C07133=1014.143,341.279,-151.610,170.583,52.042,160.243
C07134=1014.136,341.031,-151.575,170.576,52.047,160.243
C07135=1014.129,340.783,-151.540,170.568,52.051,160.243
C07136=1014.122,340.536,-151.504,170.561,52.056,160.242
C07137=1014.116,340.289,-151.469,170.554,52.060,160.242
C07138=1014.109,340.041,-151.433,170.546,52.065,160.241
C07139=1014.103,339.794,-151.398,170.539,52.069,160.241
C07140=1014.095,339.546,-151.362,170.530,52.073,160.240
C07141=1014.088,339.299,-151.326,170.523,52.077,160.240
C07142=1014.081,339.052,-151.291,170.515,52.082,160.240
C07143=1014.075,338.805,-151.256,170.508,52.086,160.239
C07144=1014.067,338.513,-151.215,170.499,52.092,160.239
C07145=1014.059,338.221,-151.173,170.490,52.097,160.239
C07146=1014.052,337.930,-151.132,170.481,52.103,160.238
C07147=1014.044,337.638,-151.090,170.472,52.108,160.238
C07148=1014.036,337.391,-151.056,170.465,52.112,160.237
C07149=1014.029,337.143,-151.021,170.457,52.117,160.237
C07150=1014.022,336.896,-150.986,170.450,52.122,160.237
C07151=1014.016,336.648,-150.951,170.442,52.127,160.236
C07152=1014.009,336.401,-150.916,170.435,52.131,160.236
C07153=1014.002,336.153,-150.881,170.426,52.136,160.236
C07154=1013.996,335.906,-150.846,170.420,52.141,160.236
C07155=1013.989,335.658,-150.811,170.412,52.146,160.235
C07156=1013.983,335.410,-150.776,170.405,52.150,160.235
C07157=1013.976,335.163,-150.741,170.397,52.154,160.234
C07158=1013.969,334.915,-150.707,170.390,52.160,160.234
C07159=1013.963,334.668,-150.672,170.383,52.164,160.234
C07160=1013.956,334.421,-150.637,170.374,52.169,160.233
C07161=1013.949,334.173,-150.603,170.368,52.174,160.233
C07162=1013.942,333.926,-150.568,170.361,52.178,160.233
C07163=1013.936,333.678,-150.533,170.353,52.183,160.233
C07164=1013.929,333.431,-150.498,170.346,52.188,160.232
C07165=1013.923,333.183,-150.464,170.338,52.192,160.232
C07166=1013.917,332.936,-150.429,170.331,52.197,160.232
C07167=1013.910,332.688,-150.395,170.324,52.202,160.232
C07168=1013.903,332.441,-150.359,170.316,52.207,160.231
C07169=1013.897,332.193,-150.325,170.309,52.211,160.231
C07170=1013.891,331.945,-150.291,170.301,52.217,160.231
C07171=1013.883,331.698,-150.256,170.294,52.221,160.230
C07172=1013.877,331.450,-150.222,170.287,52.226,160.230
C07173=1013.871,331.203,-150.188,170.280,52.231,160.230
C07174=1013.864,330.955,-150.154,170.272,52.236,160.230
C07175=1013.857,330.707,-150.120,170.265,52.241,160.230
C07176=1013.851,330.460,-150.085,170.258,52.246,160.229
C07177=1013.844,330.213,-150.051,170.251,52.251,160.229
C07178=1013.838,329.965,-150.017,170.243,52.256,160.229
C07179=1013.831,329.717,-149.982,170.236,52.261,160.229
C07180=1013.825,329.470,-149.949,170.229,52.266,160.229
C07181=1013.818,329.222,-149.914,170.222,52.271,160.228
C07182=1013.812,328.975,-149.881,170.215,52.276,160.228
C07183=1013.805,328.727,-149.847,170.207,52.281,160.228
C07184=1013.799,328.479,-149.812,170.201,52.286,160.228
C07185=1013.792,328.232,-149.779,170.194,52.291,160.228
C07186=1013.786,327.984,-149.744,170.186,52.296,160.227
C07187=1013.780,327.737,-149.710,170.179,52.301,160.227
C07188=1013.772,327.489,-149.676,170.171,52.306,160.227
C07189=1013.767,327.242,-149.642,170.165,52.311,160.227
C07190=1013.760,326.994,-149.608,170.158,52.316,160.227
C07191=1013.754,326.746,-149.575,170.150,52.322,160.226
C07192=1013.747,326.498,-149.541,170.143,52.327,160.226
C07193=1013.742,326.251,-149.507,170.137,52.332,160.226
C07194=1013.734,326.003,-149.473,170.129,52.337,160.226
C07195=1013.728,325.756,-149.439,170.122,52.342,160.226
C07196=1013.722,325.508,-149.406,170.116,52.347,160.226
C07197=1013.715,325.261,-149.372,170.108,52.352,160.225
C07198=1013.709,325.013,-149.339,170.101,52.357,160.225
C07199=1013.702,324.765,-149.305,170.093,52.363,160.225
C07200=1013.696,324.518,-149.272,170.087,52.368,160.225
C07201=1013.689,324.270,-149.239,170.080,52.374,160.225
C07202=1013.682,324.022,-149.206,170.073,52.379,160.225
C07203=1013.676,323.775,-149.171,170.066,52.384,160.225
C07204=1013.669,323.479,-149.132,170.058,52.390,160.224
C07205=1013.660,323.183,-149.093,170.050,52.397,160.224
C07206=1013.653,322.887,-149.053,170.040,52.404,160.224
C07207=1013.645,322.591,-149.013,170.032,52.410,160.224
C07208=1013.638,322.344,-148.980,170.025,52.415,160.224
C07209=1013.632,322.096,-148.947,170.019,52.421,160.224
C07210=1013.626,321.848,-148.913,170.011,52.426,160.224
C07211=1013.620,321.600,-148.880,170.005,52.431,160.224
C07212=1013.613,321.353,-148.847,169.998,52.437,160.224
C07213=1013.606,321.105,-148.814,169.991,52.442,160.224
C07214=1013.600,320.857,-148.781,169.984,52.448,160.224
C07215=1013.594,320.609,-148.748,169.977,52.453,160.223
C07216=1013.588,320.362,-148.715,169.970,52.458,160.223
C07217=1013.581,320.113,-148.682,169.964,52.464,160.223
C07218=1013.575,319.866,-148.649,169.956,52.469,160.223
C07219=1013.568,319.619,-148.616,169.950,52.475,160.223
C07220=1013.563,319.371,-148.582,169.943,52.480,160.223
C07221=1013.556,319.123,-148.550,169.936,52.486,160.223
C07222=1013.550,318.876,-148.517,169.929,52.491,160.223
C07223=1013.544,318.628,-148.484,169.922,52.497,160.223
C07224=1013.537,318.380,-148.451,169.916,52.503,160.223
C07225=1013.531,318.132,-148.418,169.909,52.508,160.223
C07226=1013.525,317.884,-148.385,169.902,52.514,160.223
C07227=1013.519,317.637,-148.352,169.895,52.519,160.223
C07228=1013.513,317.389,-148.320,169.889,52.525,160.223
C07229=1013.506,317.142,-148.287,169.881,52.531,160.223
C07230=1013.500,316.894,-148.254,169.875,52.536,160.223
C07231=1013.494,316.646,-148.221,169.869,52.542,160.223
C07232=1013.488,316.398,-148.189,169.861,52.548,160.223
C07233=1013.482,316.150,-148.156,169.855,52.553,160.223
C07234=1013.476,315.903,-148.123,169.848,52.558,160.223
C07235=1013.470,315.655,-148.090,169.841,52.564,160.223
C07236=1013.464,315.407,-148.057,169.835,52.570,160.223
C07237=1013.458,315.159,-148.025,169.829,52.576,160.223
C07238=1013.452,314.911,-147.992,169.821,52.581,160.223
C07239=1013.445,314.664,-147.960,169.815,52.587,160.223
C07240=1013.439,314.416,-147.927,169.808,52.593,160.223
C07241=1013.433,314.168,-147.895,169.801,52.599,160.223
C07242=1013.428,313.920,-147.861,169.795,52.605,160.223
C07243=1013.422,313.673,-147.829,169.788,52.610,160.223
C07244=1013.416,313.425,-147.797,169.781,52.616,160.223
C07245=1013.410,313.177,-147.764,169.775,52.621,160.223
C07246=1013.403,312.930,-147.732,169.768,52.627,160.223
C07247=1013.397,312.682,-147.700,169.761,52.633,160.223
C07248=1013.392,312.434,-147.666,169.755,52.639,160.223
C07249=1013.386,312.186,-147.635,169.749,52.645,160.223
C07250=1013.380,311.939,-147.602,169.741,52.651,160.223
C07251=1013.374,311.691,-147.569,169.735,52.656,160.223
C07252=1013.368,311.443,-147.537,169.729,52.662,160.223
C07253=1013.363,311.196,-147.504,169.723,52.668,160.223
C07254=1013.357,310.947,-147.472,169.715,52.674,160.223
C07255=1013.351,310.700,-147.439,169.709,52.680,160.223
C07256=1013.345,310.452,-147.407,169.703,52.685,160.223
C07257=1013.339,310.204,-147.376,169.696,52.691,160.223
C07258=1013.333,309.956,-147.343,169.689,52.697,160.223
C07259=1013.328,309.708,-147.310,169.683,52.703,160.223
C07260=1013.322,309.461,-147.278,169.676,52.709,160.223
C07261=1013.316,309.213,-147.246,169.670,52.715,160.224
C07262=1013.310,308.965,-147.214,169.664,52.721,160.224
C07263=1013.304,308.717,-147.183,169.657,52.727,160.224
C07264=1013.297,308.427,-147.145,169.650,52.734,160.224
C07265=1013.290,308.137,-147.109,169.642,52.741,160.224
C07266=1013.283,307.846,-147.071,169.634,52.748,160.224
C07267=1013.275,307.555,-147.034,169.627,52.756,160.225
C07268=1013.269,307.308,-147.003,169.621,52.762,160.225
C07269=1013.263,307.060,-146.971,169.613,52.768,160.225
C07270=1013.257,306.812,-146.939,169.607,52.774,160.225
C07271=1013.251,306.564,-146.908,169.600,52.781,160.225
C07272=1013.245,306.316,-146.876,169.594,52.787,160.225
C07273=1013.239,306.069,-146.845,169.588,52.793,160.225
C07274=1013.233,305.820,-146.814,169.581,52.799,160.225
C07275=1013.227,305.573,-146.782,169.575,52.805,160.225
C07276=1013.221,305.325,-146.750,169.568,52.812,160.226
C07277=1013.214,305.077,-146.719,169.562,52.818,160.226
C07278=1013.209,304.829,-146.688,169.556,52.824,160.226
C07279=1013.202,304.581,-146.657,169.549,52.830,160.226
C07280=1013.197,304.333,-146.625,169.543,52.837,160.226
C07281=1013.190,304.085,-146.594,169.536,52.843,160.226
C07282=1013.185,303.837,-146.563,169.530,52.849,160.227
C07283=1013.178,303.589,-146.531,169.524,52.856,160.227
C07284=1013.173,303.342,-146.499,169.517,52.862,160.227
C07285=1013.167,303.093,-146.469,169.511,52.868,160.227
C07286=1013.161,302.846,-146.437,169.505,52.875,160.227
C07287=1013.155,302.597,-146.406,169.498,52.881,160.227
C07288=1013.149,302.350,-146.375,169.493,52.887,160.228
C07289=1013.144,302.102,-146.344,169.486,52.894,160.228
C07290=1013.138,301.854,-146.312,169.480,52.900,160.228
C07291=1013.131,301.607,-146.281,169.474,52.906,160.228
C07292=1013.126,301.358,-146.250,169.467,52.913,160.228
C07293=1013.120,301.110,-146.218,169.461,52.919,160.229
C07294=1013.115,300.862,-146.188,169.454,52.926,160.229
C07295=1013.109,300.614,-146.157,169.448,52.932,160.229
C07296=1013.103,300.366,-146.126,169.442,52.938,160.229
C07297=1013.098,300.118,-146.095,169.436,52.945,160.230
C07298=1013.091,299.870,-146.063,169.430,52.952,160.230
C07299=1013.086,299.622,-146.032,169.423,52.958,160.230
C07300=1013.080,299.374,-146.002,169.417,52.964,160.230
C07301=1013.074,299.126,-145.970,169.411,52.971,160.230
C07302=1013.068,298.878,-145.940,169.404,52.977,160.231
C07303=1013.063,298.631,-145.908,169.398,52.984,160.231
C07304=1013.057,298.383,-145.878,169.393,52.990,160.231
C07305=1013.051,298.134,-145.846,169.386,52.997,160.231
C07306=1013.046,297.886,-145.816,169.380,53.004,160.232
C07307=1013.040,297.639,-145.784,169.373,53.010,160.232
C07308=1013.034,297.391,-145.754,169.368,53.017,160.232
C07309=1013.029,297.142,-145.723,169.362,53.023,160.232
C07310=1013.023,296.894,-145.692,169.355,53.030,160.233
C07311=1013.017,296.647,-145.661,169.349,53.037,160.233
C07312=1013.012,296.399,-145.630,169.344,53.043,160.233
C07313=1013.007,296.151,-145.599,169.337,53.050,160.233
C07314=1013.000,295.902,-145.569,169.331,53.056,160.234
C07315=1012.995,295.654,-145.538,169.325,53.063,160.234
C07316=1012.989,295.406,-145.507,169.318,53.070,160.234
C07317=1012.984,295.158,-145.476,169.313,53.076,160.234
C07318=1012.978,294.911,-145.446,169.306,53.083,160.235
C07319=1012.973,294.663,-145.414,169.300,53.089,160.235
C07320=1012.967,294.415,-145.384,169.294,53.096,160.235
C07321=1012.962,294.167,-145.353,169.288,53.103,160.235
C07322=1012.956,293.919,-145.323,169.282,53.109,160.236
C07323=1012.951,293.671,-145.292,169.276,53.116,160.236
C07324=1012.945,293.398,-145.258,169.269,53.123,160.236
C07325=1012.939,293.126,-145.224,169.262,53.131,160.237
C07326=1012.933,292.853,-145.190,169.256,53.138,160.237
C07327=1012.927,292.582,-145.157,169.249,53.145,160.237
C07328=1012.922,292.334,-145.126,169.243,53.153,160.238
C07329=1012.916,292.085,-145.097,169.237,53.159,160.238
C07330=1012.911,291.837,-145.066,169.231,53.166,160.238
C07331=1012.905,291.590,-145.036,169.225,53.173,160.239
C07332=1012.899,291.342,-145.006,169.219,53.180,160.239
C07333=1012.894,291.093,-144.976,169.213,53.187,160.239
C07334=1012.888,290.845,-144.945,169.207,53.194,160.240
C07335=1012.883,290.597,-144.915,169.200,53.201,160.240
C07336=1012.877,290.349,-144.885,169.195,53.208,160.240
C07337=1012.871,290.101,-144.855,169.189,53.214,160.241
C07338=1012.866,289.853,-144.825,169.183,53.222,160.241
C07339=1012.860,289.605,-144.795,169.177,53.228,160.241
C07340=1012.854,289.356,-144.765,169.171,53.236,160.242
C07341=1012.849,289.109,-144.735,169.165,53.242,160.242
C07342=1012.843,288.860,-144.705,169.159,53.250,160.242
C07343=1012.837,288.612,-144.675,169.153,53.256,160.243
C07344=1012.832,288.364,-144.645,169.147,53.264,160.243
C07345=1012.826,288.115,-144.616,169.141,53.270,160.243
C07346=1012.821,287.868,-144.586,169.135,53.278,160.244
C07347=1012.816,287.620,-144.556,169.130,53.285,160.244
C07348=1012.810,287.372,-144.526,169.124,53.292,160.245
C07349=1012.804,287.124,-144.496,169.118,53.299,160.245
C07350=1012.799,286.875,-144.466,169.112,53.306,160.245
C07351=1012.793,286.627,-144.436,169.105,53.313,160.246
C07352=1012.787,286.379,-144.406,169.100,53.320,160.246
C07353=1012.782,286.131,-144.377,169.094,53.328,160.247
C07354=1012.777,285.883,-144.347,169.088,53.334,160.247
C07355=1012.771,285.635,-144.317,169.082,53.342,160.247
C07356=1012.766,285.386,-144.287,169.077,53.349,160.248
C07357=1012.760,285.138,-144.258,169.070,53.356,160.248
C07358=1012.755,284.890,-144.229,169.065,53.363,160.248
C07359=1012.750,284.642,-144.199,169.058,53.371,160.249
C07360=1012.744,284.393,-144.169,169.053,53.378,160.249
C07361=1012.738,284.146,-144.139,169.047,53.385,160.250
C07362=1012.733,283.898,-144.110,169.041,53.392,160.250
C07363=1012.727,283.650,-144.081,169.035,53.400,160.250
C07364=1012.722,283.401,-144.051,169.029,53.407,160.251
C07365=1012.717,283.154,-144.022,169.023,53.414,160.251
C07366=1012.711,282.905,-143.993,169.018,53.421,160.252
C07367=1012.705,282.657,-143.963,169.012,53.429,160.252
C07368=1012.700,282.408,-143.934,169.006,53.436,160.253
C07369=1012.694,282.160,-143.905,169.000,53.444,160.253
C07370=1012.689,281.912,-143.876,168.995,53.451,160.254
C07371=1012.683,281.664,-143.846,168.988,53.459,160.254
C07372=1012.678,281.416,-143.817,168.983,53.466,160.255
C07373=1012.672,281.168,-143.788,168.977,53.473,160.255
C07374=1012.666,280.919,-143.758,168.972,53.481,160.255
C07375=1012.662,280.671,-143.730,168.965,53.488,160.256
C07376=1012.656,280.423,-143.701,168.960,53.495,160.256
C07377=1012.651,280.175,-143.671,168.954,53.503,160.257
C07378=1012.645,279.927,-143.642,168.948,53.510,160.257
C07379=1012.640,279.678,-143.613,168.942,53.518,160.258
C07380=1012.634,279.430,-143.584,168.936,53.525,160.258
C07381=1012.629,279.182,-143.555,168.931,53.533,160.259
C07382=1012.624,278.934,-143.525,168.924,53.540,160.259
C07383=1012.618,278.685,-143.497,168.920,53.548,160.260
C07384=1012.612,278.425,-143.466,168.913,53.556,160.260
C07385=1012.607,278.165,-143.435,168.907,53.563,160.260
C07386=1012.602,277.905,-143.405,168.901,53.572,160.261
C07387=1012.596,277.645,-143.374,168.895,53.579,160.261
C07388=1012.587,277.237,-143.328,168.886,53.592,160.262
C07389=1012.579,276.829,-143.280,168.877,53.604,160.263
C07390=1012.570,276.422,-143.232,168.867,53.617,160.264
C07391=1012.561,276.014,-143.184,168.858,53.629,160.265
C07392=1012.347,278.241,-143.809,168.878,53.661,160.276
C07393=1012.354,278.605,-143.851,168.887,53.650,160.276
C07394=1012.362,278.970,-143.893,168.895,53.639,160.275
C07395=1012.370,279.335,-143.936,168.904,53.628,160.274
C07396=1012.379,279.699,-143.979,168.912,53.617,160.274
C07397=1012.383,279.947,-144.008,168.918,53.609,160.273
C07398=1012.389,280.196,-144.037,168.923,53.602,160.273
C07399=1012.394,280.443,-144.066,168.929,53.594,160.272
C07400=1012.400,280.692,-144.096,168.936,53.587,160.272
C07401=1012.404,280.940,-144.124,168.941,53.580,160.271
C07402=1012.410,281.189,-144.154,168.947,53.572,160.271
C07403=1012.416,281.437,-144.183,168.952,53.565,160.270
C07404=1012.421,281.684,-144.212,168.959,53.557,160.270
C07405=1012.426,281.934,-144.241,168.964,53.550,160.270
C07406=1012.433,282.182,-144.270,168.970,53.542,160.269
C07407=1012.437,282.429,-144.299,168.977,53.535,160.269
C07408=1012.443,282.678,-144.329,168.982,53.528,160.268
C07409=1012.448,282.926,-144.359,168.988,53.520,160.268
C07410=1012.454,283.174,-144.387,168.993,53.513,160.267
C07411=1012.460,283.422,-144.417,169.000,53.505,160.267
C07412=1012.465,283.671,-144.447,169.005,53.498,160.266
C07413=1012.471,283.918,-144.475,169.011,53.490,160.266
C07414=1012.476,284.166,-144.505,169.016,53.483,160.266
C07415=1012.482,284.415,-144.534,169.023,53.476,160.265
C07416=1012.487,284.663,-144.564,169.028,53.469,160.265
C07417=1012.492,284.911,-144.593,169.035,53.462,160.264
C07418=1012.498,285.160,-144.623,169.040,53.454,160.264
C07419=1012.503,285.408,-144.653,169.047,53.447,160.264
C07420=1012.508,285.656,-144.682,169.052,53.440,160.263
C07421=1012.514,285.904,-144.712,169.058,53.433,160.263
C07422=1012.519,286.152,-144.742,169.065,53.425,160.263
C07423=1012.525,286.400,-144.772,169.070,53.419,160.262
C07424=1012.530,286.648,-144.801,169.077,53.411,160.262
C07425=1012.535,286.897,-144.830,169.082,53.404,160.261
C07426=1012.541,287.144,-144.861,169.089,53.397,160.261
C07427=1012.547,287.393,-144.890,169.094,53.390,160.261
C07428=1012.552,287.641,-144.920,169.100,53.382,160.260
C07429=1012.558,287.889,-144.950,169.106,53.376,160.260
C07430=1012.563,288.137,-144.980,169.112,53.368,160.260
C07431=1012.568,288.385,-145.009,169.118,53.362,160.259
C07432=1012.574,288.633,-145.040,169.124,53.354,160.259
C07433=1012.580,288.882,-145.069,169.129,53.347,160.258
C07434=1012.585,289.130,-145.099,169.136,53.340,160.258
C07435=1012.591,289.378,-145.129,169.141,53.333,160.258
C07436=1012.597,289.626,-145.159,169.148,53.326,160.258
C07437=1012.602,289.874,-145.189,169.154,53.319,160.257
C07438=1012.607,290.122,-145.219,169.160,53.312,160.257
C07439=1012.613,290.370,-145.249,169.166,53.305,160.256
C07440=1012.619,290.618,-145.279,169.172,53.298,160.256
C07441=1012.625,290.866,-145.309,169.178,53.291,160.256
C07442=1012.630,291.114,-145.339,169.183,53.284,160.255
C07443=1012.635,291.362,-145.369,169.190,53.277,160.255
C07444=1012.641,291.610,-145.400,169.195,53.270,160.255
C07445=1012.646,291.859,-145.429,169.202,53.263,160.254
C07446=1012.652,292.107,-145.460,169.207,53.256,160.254
C07447=1012.658,292.354,-145.490,169.214,53.249,160.254
C07448=1012.663,292.603,-145.521,169.220,53.243,160.253
C07449=1012.669,292.877,-145.555,169.227,53.235,160.253
C07450=1012.676,293.152,-145.588,169.234,53.227,160.253
C07451=1012.681,293.426,-145.622,169.240,53.220,160.253
C07452=1012.688,293.701,-145.656,169.248,53.213,160.252
C07453=1012.693,293.949,-145.687,169.253,53.206,160.252
C07454=1012.699,294.197,-145.717,169.259,53.199,160.251
C07455=1012.704,294.445,-145.748,169.265,53.192,160.251
C07456=1012.710,294.693,-145.779,169.271,53.186,160.251
C07457=1012.715,294.941,-145.810,169.278,53.179,160.251
C07458=1012.720,295.189,-145.840,169.284,53.172,160.251
C07459=1012.726,295.437,-145.871,169.290,53.166,160.250
C07460=1012.731,295.685,-145.901,169.296,53.159,160.250
C07461=1012.736,295.933,-145.932,169.302,53.153,160.250
C07462=1012.742,296.181,-145.963,169.309,53.146,160.250
C07463=1012.747,296.429,-145.994,169.314,53.139,160.249
C07464=1012.754,296.677,-146.024,169.321,53.132,160.249
C07465=1012.759,296.925,-146.056,169.327,53.125,160.249
C07466=1012.765,297.173,-146.086,169.332,53.119,160.248
C07467=1012.770,297.421,-146.117,169.339,53.112,160.248
C07468=1012.775,297.669,-146.148,169.345,53.105,160.248
C07469=1012.781,297.917,-146.179,169.352,53.099,160.248
C07470=1012.787,298.165,-146.211,169.357,53.092,160.247
C07471=1012.793,298.413,-146.241,169.364,53.086,160.247
C07472=1012.798,298.661,-146.272,169.370,53.080,160.247
C07473=1012.804,298.909,-146.302,169.376,53.073,160.247
C07474=1012.810,299.157,-146.334,169.383,53.066,160.247
C07475=1012.815,299.405,-146.365,169.389,53.060,160.246
C07476=1012.820,299.653,-146.396,169.396,53.053,160.246
C07477=1012.827,299.900,-146.427,169.401,53.047,160.246
C07478=1012.832,300.149,-146.458,169.407,53.040,160.246
C07479=1012.838,300.397,-146.488,169.414,53.033,160.245
C07480=1012.843,300.644,-146.520,169.420,53.027,160.245
C07481=1012.850,300.893,-146.551,169.427,53.021,160.245
C07482=1012.855,301.140,-146.582,169.433,53.014,160.245
C07483=1012.861,301.388,-146.613,169.439,53.007,160.245
C07484=1012.867,301.637,-146.644,169.445,53.001,160.244
C07485=1012.873,301.884,-146.675,169.451,52.995,160.244
C07486=1012.878,302.132,-146.706,169.458,52.988,160.244
C07487=1012.885,302.380,-146.737,169.464,52.982,160.244
C07488=1012.890,302.628,-146.768,169.471,52.976,160.244
C07489=1012.897,302.876,-146.800,169.477,52.969,160.244
C07490=1012.902,303.124,-146.831,169.484,52.962,160.243
C07491=1012.908,303.372,-146.862,169.490,52.956,160.243
C07492=1012.914,303.620,-146.894,169.497,52.950,160.243
C07493=1012.920,303.868,-146.924,169.503,52.943,160.243
C07494=1012.926,304.116,-146.956,169.509,52.938,160.243
C07495=1012.932,304.363,-146.987,169.516,52.931,160.243
C07496=1012.937,304.612,-147.019,169.521,52.924,160.242
C07497=1012.943,304.859,-147.050,169.529,52.918,160.242
C07498=1012.949,305.107,-147.082,169.534,52.912,160.242
C07499=1012.955,305.355,-147.113,169.542,52.906,160.242
C07500=1012.961,305.603,-147.144,169.547,52.899,160.242
C07501=1012.967,305.851,-147.176,169.554,52.893,160.242
C07502=1012.973,306.099,-147.207,169.560,52.887,160.242
C07503=1012.979,306.348,-147.238,169.566,52.880,160.241
C07504=1012.985,306.595,-147.270,169.573,52.874,160.241
C07505=1012.991,306.843,-147.302,169.579,52.868,160.241
C07506=1012.997,307.090,-147.333,169.586,52.862,160.241
C07507=1013.003,307.338,-147.365,169.593,52.856,160.241
C07508=1013.010,307.587,-147.395,169.599,52.849,160.241
C07509=1013.016,307.879,-147.434,169.607,52.842,160.241
C07510=1013.024,308.172,-147.470,169.615,52.835,160.241
C07511=1013.031,308.464,-147.507,169.623,52.828,160.240
C07512=1013.038,308.757,-147.544,169.630,52.820,160.240
C07513=1013.044,309.004,-147.577,169.636,52.814,160.240
C07514=1013.050,309.252,-147.609,169.643,52.808,160.240
C07515=1013.056,309.501,-147.641,169.650,52.802,160.240
C07516=1013.061,309.748,-147.673,169.656,52.796,160.240
C07517=1013.068,309.996,-147.705,169.663,52.790,160.240
C07518=1013.072,310.244,-147.738,169.669,52.784,160.240
C07519=1013.079,310.491,-147.770,169.675,52.778,160.240
C07520=1013.085,310.739,-147.802,169.683,52.772,160.240
C07521=1013.090,310.987,-147.834,169.689,52.766,160.240
C07522=1013.096,311.235,-147.867,169.695,52.761,160.239
C07523=1013.102,311.483,-147.899,169.702,52.754,160.239
C07524=1013.108,311.731,-147.932,169.709,52.749,160.239
C07525=1013.113,311.978,-147.964,169.715,52.743,160.239
C07526=1013.120,312.226,-147.996,169.722,52.737,160.239
C07527=1013.126,312.474,-148.029,169.728,52.731,160.239
C07528=1013.132,312.722,-148.061,169.735,52.725,160.239
C07529=1013.137,312.969,-148.093,169.742,52.719,160.239
C07530=1013.143,313.217,-148.126,169.748,52.714,160.239
C07531=1013.149,313.465,-148.159,169.755,52.708,160.239
C07532=1013.155,313.713,-148.191,169.762,52.702,160.239
C07533=1013.161,313.960,-148.224,169.768,52.696,160.239
C07534=1013.168,314.208,-148.257,169.775,52.690,160.239
C07535=1013.173,314.455,-148.288,169.781,52.684,160.239
C07536=1013.179,314.703,-148.322,169.789,52.678,160.239
C07537=1013.185,314.951,-148.354,169.795,52.673,160.239
C07538=1013.191,315.199,-148.386,169.802,52.667,160.239
C07539=1013.197,315.447,-148.419,169.809,52.661,160.239
C07540=1013.203,315.694,-148.452,169.815,52.656,160.239
C07541=1013.209,315.942,-148.485,169.821,52.650,160.239
C07542=1013.215,316.190,-148.517,169.829,52.644,160.239
C07543=1013.221,316.438,-148.550,169.835,52.639,160.239
C07544=1013.228,316.686,-148.583,169.842,52.633,160.239
C07545=1013.234,316.933,-148.615,169.849,52.627,160.239
C07546=1013.240,317.181,-148.648,169.855,52.622,160.239
C07547=1013.246,317.429,-148.681,169.863,52.616,160.239
C07548=1013.252,317.677,-148.713,169.869,52.610,160.239
C07549=1013.258,317.925,-148.746,169.877,52.605,160.239
C07550=1013.264,318.172,-148.779,169.883,52.599,160.239
C07551=1013.271,318.420,-148.812,169.890,52.593,160.239
C07552=1013.276,318.668,-148.845,169.897,52.588,160.239
C07553=1013.282,318.915,-148.878,169.903,52.582,160.239
C07554=1013.289,319.163,-148.911,169.910,52.576,160.239
C07555=1013.296,319.411,-148.944,169.917,52.571,160.239
C07556=1013.302,319.659,-148.976,169.924,52.565,160.239
C07557=1013.307,319.907,-149.010,169.931,52.560,160.240
C07558=1013.314,320.154,-149.042,169.937,52.554,160.239
C07559=1013.320,320.401,-149.076,169.945,52.549,160.240
C07560=1013.327,320.649,-149.109,169.951,52.543,160.240
C07561=1013.334,320.897,-149.142,169.959,52.538,160.240
C07562=1013.339,321.145,-149.175,169.965,52.532,160.240
C07563=1013.345,321.393,-149.208,169.973,52.526,160.240
C07564=1013.352,321.640,-149.241,169.979,52.521,160.240
C07565=1013.359,321.888,-149.274,169.987,52.515,160.240
C07566=1013.365,322.135,-149.307,169.993,52.510,160.240
C07567=1013.371,322.383,-149.340,170.000,52.505,160.240
C07568=1013.377,322.631,-149.373,170.007,52.499,160.240
C07569=1013.385,322.929,-149.413,170.016,52.493,160.241
C07570=1013.393,323.227,-149.453,170.024,52.486,160.241
C07571=1013.401,323.525,-149.493,170.032,52.480,160.241
C07572=1013.409,323.824,-149.533,170.041,52.473,160.241
C07573=1013.415,324.072,-149.567,170.048,52.468,160.241
C07574=1013.421,324.319,-149.600,170.055,52.462,160.241
C07575=1013.428,324.567,-149.633,170.062,52.457,160.241
C07576=1013.435,324.814,-149.666,170.070,52.451,160.241
C07577=1013.441,325.061,-149.699,170.076,52.446,160.242
C07578=1013.447,325.310,-149.733,170.083,52.441,160.241
C07579=1013.454,325.557,-149.767,170.090,52.435,160.242
C07580=1013.461,325.805,-149.800,170.097,52.430,160.242
C07581=1013.467,326.053,-149.834,170.105,52.425,160.242
C07582=1013.473,326.300,-149.868,170.112,52.420,160.242
C07583=1013.480,326.548,-149.902,170.119,52.414,160.242
C07584=1013.486,326.795,-149.936,170.126,52.409,160.243
C07585=1013.493,327.043,-149.969,170.133,52.404,160.243
C07586=1013.498,327.290,-150.003,170.140,52.399,160.243
C07587=1013.505,327.538,-150.037,170.147,52.394,160.243
C07588=1013.511,327.785,-150.071,170.155,52.389,160.243
C07589=1013.518,328.033,-150.105,170.161,52.384,160.243
C07590=1013.524,328.281,-150.139,170.169,52.378,160.244
C07591=1013.531,328.528,-150.173,170.176,52.373,160.244
C07592=1013.537,328.776,-150.207,170.183,52.369,160.244
C07593=1013.543,329.024,-150.242,170.191,52.363,160.244
C07594=1013.551,329.271,-150.275,170.197,52.358,160.244
C07595=1013.556,329.519,-150.309,170.205,52.353,160.245
C07596=1013.563,329.767,-150.344,170.212,52.348,160.245
C07597=1013.569,330.014,-150.377,170.219,52.343,160.245
C07598=1013.576,330.262,-150.412,170.227,52.338,160.245
C07599=1013.582,330.509,-150.446,170.234,52.333,160.246
C07600=1013.589,330.756,-150.480,170.241,52.328,160.246
C07601=1013.595,331.004,-150.514,170.249,52.322,160.246
C07602=1013.602,331.252,-150.548,170.256,52.318,160.246
C07603=1013.609,331.499,-150.583,170.264,52.313,160.247
C07604=1013.615,331.747,-150.617,170.270,52.308,160.247
C07605=1013.622,331.995,-150.651,170.277,52.303,160.247
C07606=1013.628,332.243,-150.686,170.285,52.298,160.247
C07607=1013.635,332.489,-150.720,170.292,52.294,160.248
C07608=1013.642,332.737,-150.754,170.300,52.288,160.248
C07609=1013.648,332.984,-150.790,170.307,52.283,160.248
C07610=1013.655,333.232,-150.824,170.315,52.279,160.248
C07611=1013.661,333.480,-150.858,170.321,52.274,160.248
C07612=1013.667,333.727,-150.893,170.330,52.269,160.249
C07613=1013.674,333.975,-150.928,170.337,52.264,160.249
C07614=1013.681,334.222,-150.963,170.344,52.259,160.249
C07615=1013.687,334.470,-150.997,170.352,52.255,160.250
C07616=1013.694,334.718,-151.032,170.358,52.250,160.250
C07617=1013.700,334.964,-151.067,170.366,52.245,160.250
C07618=1013.707,335.212,-151.101,170.373,52.240,160.250
C07619=1013.714,335.459,-151.136,170.381,52.235,160.251
C07620=1013.720,335.707,-151.170,170.388,52.231,160.251
C07621=1013.727,335.955,-151.206,170.396,52.226,160.251
C07622=1013.734,336.202,-151.241,170.403,52.221,160.252
C07623=1013.740,336.450,-151.275,170.411,52.217,160.252
C07624=1013.747,336.698,-151.310,170.418,52.212,160.253
C07625=1013.754,336.945,-151.345,170.426,52.207,160.253
C07626=1013.761,337.192,-151.381,170.433,52.202,160.253
C07627=1013.768,337.440,-151.416,170.441,52.198,160.254
C07628=1013.774,337.688,-151.450,170.449,52.193,160.254
C07629=1013.782,337.981,-151.491,170.458,52.187,160.254
C07630=1013.790,338.275,-151.533,170.467,52.182,160.255
C07631=1013.798,338.568,-151.575,170.476,52.176,160.255
C07632=1013.807,338.863,-151.617,170.485,52.171,160.256
C07633=1013.813,339.110,-151.652,170.492,52.167,160.256
C07634=1013.819,339.358,-151.688,170.500,52.162,160.256
C07635=1013.826,339.605,-151.723,170.507,52.157,160.257
C07636=1013.833,339.852,-151.758,170.515,52.153,160.257
C07637=1013.840,340.100,-151.793,170.522,52.148,160.257
C07638=1013.847,340.347,-151.828,170.531,52.144,160.258
C07639=1013.854,340.594,-151.864,170.538,52.140,160.258
C07640=1013.860,340.842,-151.900,170.546,52.135,160.259
C07641=1013.867,341.090,-151.935,170.554,52.130,160.259
C07642=1013.874,341.337,-151.970,170.562,52.126,160.260
C07643=1013.881,341.584,-152.006,170.570,52.121,160.260
C07644=1013.888,341.831,-152.041,170.577,52.117,160.260
C07645=1013.894,342.079,-152.077,170.585,52.112,160.261
C07646=1013.901,342.326,-152.113,170.593,52.109,160.261
C07647=1013.908,342.574,-152.148,170.601,52.104,160.262
C07648=1013.915,342.821,-152.184,170.608,52.100,160.262
C07649=1013.922,343.069,-152.220,170.616,52.095,160.262
C07650=1013.929,343.316,-152.256,170.624,52.091,160.263
C07651=1013.936,343.563,-152.291,170.632,52.086,160.263
C07652=1013.942,343.810,-152.327,170.640,52.082,160.264
C07653=1013.949,344.058,-152.363,170.647,52.078,160.264
C07654=1013.956,344.305,-152.398,170.656,52.073,160.265
C07655=1013.963,344.552,-152.434,170.663,52.069,160.265
C07656=1013.971,344.799,-152.471,170.671,52.065,160.266
C07657=1013.977,345.047,-152.506,170.678,52.061,160.266
C07658=1013.985,345.295,-152.542,170.686,52.056,160.267
C07659=1013.992,345.541,-152.578,170.695,52.052,160.267
C07660=1013.998,345.789,-152.613,170.702,52.048,160.268
C07661=1014.005,346.036,-152.650,170.711,52.044,160.268
C07662=1014.012,346.283,-152.686,170.718,52.039,160.269
C07663=1014.020,346.531,-152.722,170.726,52.035,160.269
C07664=1014.026,346.778,-152.758,170.735,52.030,160.270
C07665=1014.034,347.026,-152.794,170.742,52.027,160.270
C07666=1014.040,347.273,-152.831,170.751,52.023,160.271
C07667=1014.048,347.520,-152.867,170.758,52.018,160.271
C07668=1014.054,347.767,-152.903,170.766,52.014,160.272
C07669=1014.062,348.015,-152.940,170.775,52.010,160.272
C07670=1014.068,348.262,-152.976,170.782,52.006,160.273
C07671=1014.076,348.509,-153.012,170.791,52.002,160.273
C07672=1014.082,348.756,-153.049,170.799,51.998,160.274
C07673=1014.090,349.004,-153.085,170.807,51.994,160.275
C07674=1014.097,349.251,-153.122,170.815,51.989,160.275
C07675=1014.104,349.498,-153.158,170.823,51.986,160.276
C07676=1014.111,349.745,-153.195,170.831,51.982,160.276
C07677=1014.118,349.992,-153.231,170.840,51.978,160.277
C07678=1014.125,350.240,-153.268,170.847,51.974,160.277
C07679=1014.133,350.487,-153.305,170.856,51.970,160.278
C07680=1014.139,350.734,-153.341,170.864,51.966,160.279
C07681=1014.147,350.981,-153.377,170.871,51.962,160.279
C07682=1014.154,351.229,-153.414,170.880,51.958,160.280
C07683=1014.161,351.476,-153.452,170.889,51.954,160.280
C07684=1014.168,351.723,-153.488,170.896,51.950,160.281
C07685=1014.175,351.971,-153.524,170.905,51.946,160.281
C07686=1014.183,352.217,-153.561,170.913,51.942,160.282
C07687=1014.190,352.465,-153.598,170.922,51.938,160.283
C07688=1014.198,352.711,-153.635,170.929,51.934,160.283
C07689=1014.206,353.003,-153.679,170.940,51.929,160.284
C07690=1014.215,353.294,-153.722,170.950,51.925,160.285
C07691=1014.223,353.586,-153.766,170.959,51.920,160.286
C07692=1014.232,353.877,-153.809,170.969,51.916,160.286
C07693=1014.239,354.124,-153.846,170.978,51.913,160.287
C07694=1014.246,354.372,-153.883,170.986,51.908,160.288
C07695=1014.254,354.618,-153.920,170.994,51.905,160.288
C07696=1014.261,354.865,-153.957,171.002,51.901,160.289
C07697=1014.268,355.112,-153.995,171.011,51.897,160.290
C07698=1014.275,355.359,-154.032,171.020,51.893,160.290
C07699=1014.283,355.607,-154.069,171.027,51.890,160.291
C07700=1014.290,355.854,-154.106,171.036,51.886,160.292
C07701=1014.298,356.101,-154.144,171.045,51.882,160.292
C07702=1014.306,356.348,-154.181,171.053,51.878,160.293
C07703=1014.313,356.595,-154.218,171.061,51.875,160.294
C07704=1014.320,356.842,-154.256,171.070,51.871,160.294
C07705=1014.327,357.089,-154.293,171.079,51.868,160.295
C07706=1014.335,357.336,-154.331,171.088,51.864,160.296
C07707=1014.343,357.583,-154.368,171.097,51.860,160.297
C07708=1014.350,357.831,-154.405,171.104,51.857,160.297
C07709=1014.358,358.078,-154.443,171.113,51.853,160.298
C07710=1014.365,358.325,-154.481,171.122,51.850,160.299
C07711=1014.373,358.571,-154.518,171.131,51.846,160.300
C07712=1014.380,358.818,-154.556,171.140,51.842,160.301
C07713=1014.388,359.066,-154.593,171.147,51.839,160.301
C07714=1014.395,359.312,-154.631,171.156,51.835,160.302
C07715=1014.402,359.559,-154.669,171.165,51.832,160.303
C07716=1014.410,359.807,-154.707,171.174,51.828,160.304
C07717=1014.417,360.054,-154.746,171.183,51.824,160.304
C07718=1014.424,360.301,-154.783,171.191,51.821,160.305
C07719=1014.432,360.548,-154.821,171.200,51.818,160.306
C07720=1014.439,360.795,-154.859,171.209,51.815,160.307
C07721=1014.447,361.042,-154.898,171.218,51.811,160.308
C07722=1014.455,361.289,-154.935,171.227,51.808,160.308
C07723=1014.462,361.536,-154.973,171.236,51.804,160.309
C07724=1014.470,361.782,-155.012,171.243,51.801,160.310
C07725=1014.478,362.030,-155.050,171.252,51.797,160.311
C07726=1014.485,362.276,-155.088,171.261,51.794,160.311
C07727=1014.493,362.523,-155.126,171.270,51.790,160.312
C07728=1014.500,362.771,-155.164,171.279,51.787,160.313
C07729=1014.508,363.017,-155.202,171.288,51.784,160.314
C07730=1014.516,363.264,-155.241,171.297,51.780,160.315
C07731=1014.524,363.511,-155.279,171.306,51.777,160.316
C07732=1014.531,363.758,-155.317,171.315,51.774,160.317
C07733=1014.539,364.005,-155.355,171.324,51.771,160.318
C07734=1014.547,364.252,-155.393,171.332,51.768,160.318
C07735=1014.555,364.499,-155.432,171.341,51.764,160.319
C07736=1014.562,364.746,-155.470,171.350,51.761,160.320
C07737=1014.571,364.993,-155.509,171.359,51.757,160.321
C07738=1014.578,365.239,-155.547,171.369,51.755,160.322
C07739=1014.586,365.487,-155.586,171.378,51.751,160.323
C07740=1014.593,365.733,-155.625,171.387,51.748,160.324
C07741=1014.601,365.981,-155.663,171.396,51.745,160.325
C07742=1014.609,366.228,-155.702,171.405,51.742,160.325
C07743=1014.617,366.474,-155.740,171.414,51.738,160.326
C07744=1014.625,366.722,-155.779,171.423,51.735,160.327
C07745=1014.633,366.967,-155.818,171.432,51.732,160.328
C07746=1014.641,367.215,-155.856,171.441,51.729,160.329
C07747=1014.649,367.462,-155.895,171.451,51.726,160.330
C07748=1014.656,367.708,-155.934,171.460,51.722,160.331
C07749=1014.666,368.007,-155.981,171.471,51.719,160.332
C07750=1014.675,368.306,-156.029,171.482,51.715,160.333
C07751=1014.685,368.605,-156.075,171.494,51.712,160.335
C07752=1014.694,368.903,-156.124,171.505,51.708,160.336
C07753=1014.702,369.151,-156.162,171.514,51.705,160.337
C07754=1014.711,369.397,-156.202,171.524,51.702,160.338
C07755=1014.718,369.643,-156.241,171.533,51.699,160.339
C07756=1014.726,369.891,-156.280,171.542,51.696,160.340
C07757=1014.734,370.138,-156.320,171.551,51.693,160.341
C07758=1014.742,370.384,-156.359,171.561,51.690,160.342
C07759=1014.750,370.631,-156.398,171.570,51.688,160.343
C07760=1014.758,370.878,-156.438,171.580,51.684,160.344
C07761=1014.766,371.124,-156.476,171.590,51.681,160.345
C07762=1014.775,371.371,-156.516,171.599,51.678,160.346
C07763=1014.782,371.618,-156.556,171.608,51.676,160.347
C07764=1014.790,371.865,-156.594,171.618,51.673,160.348
C07765=1014.798,372.112,-156.634,171.627,51.670,160.349
C07766=1014.807,372.358,-156.674,171.636,51.667,160.350
C07767=1014.815,372.605,-156.713,171.646,51.664,160.351
C07768=1014.823,372.852,-156.753,171.656,51.661,160.352
C07769=1014.831,373.099,-156.792,171.666,51.658,160.353
C07770=1014.840,373.345,-156.831,171.675,51.656,160.354
C07771=1014.847,373.592,-156.871,171.684,51.653,160.356
C07772=1014.856,373.838,-156.911,171.694,51.650,160.357
C07773=1014.864,374.085,-156.951,171.704,51.647,160.358
C07774=1014.872,374.331,-156.991,171.714,51.644,160.359
C07775=1014.881,374.578,-157.030,171.723,51.642,160.360
C07776=1014.889,374.826,-157.070,171.733,51.639,160.361
C07777=1014.898,375.072,-157.110,171.743,51.636,160.362
C07778=1014.906,375.319,-157.150,171.753,51.633,160.363
C07779=1014.914,375.565,-157.190,171.762,51.631,160.365
C07780=1014.922,375.811,-157.230,171.772,51.628,160.366
C07781=1014.930,376.058,-157.270,171.782,51.625,160.367
C07782=1014.939,376.305,-157.311,171.792,51.623,160.368
C07783=1014.947,376.552,-157.350,171.801,51.620,160.369
C07784=1014.955,376.798,-157.391,171.811,51.618,160.370
C07785=1014.963,377.044,-157.432,171.822,51.615,160.372
C07786=1014.971,377.291,-157.471,171.831,51.613,160.373
C07787=1014.980,377.538,-157.512,171.841,51.610,160.374
C07788=1014.988,377.784,-157.553,171.852,51.607,160.375
C07789=1014.997,378.030,-157.593,171.861,51.605,160.376
C07790=1015.005,378.278,-157.633,171.871,51.603,160.378
C07791=1015.013,378.524,-157.674,171.882,51.600,160.379
C07792=1015.021,378.771,-157.714,171.891,51.598,160.380
C07793=1015.031,379.017,-157.755,171.901,51.595,160.381
C07794=1015.039,379.263,-157.795,171.911,51.592,160.383
C07795=1015.047,379.510,-157.836,171.921,51.590,160.384
C07796=1015.056,379.756,-157.876,171.931,51.588,160.385
C07797=1015.064,380.003,-157.917,171.941,51.585,160.386
C07798=1015.073,380.250,-157.958,171.951,51.583,160.387
C07799=1015.081,380.496,-157.999,171.962,51.580,160.389
C07800=1015.090,380.743,-158.039,171.972,51.578,160.390
C07801=1015.098,380.989,-158.080,171.983,51.576,160.391
C07802=1015.107,381.236,-158.121,171.992,51.573,160.393
C07803=1015.116,381.482,-158.162,172.002,51.571,160.394
C07804=1015.124,381.728,-158.202,172.013,51.569,160.395
C07805=1015.133,381.975,-158.243,172.023,51.567,160.397
C07806=1015.141,382.222,-158.284,172.034,51.564,160.398
C07807=1015.151,382.468,-158.325,172.043,51.562,160.399
C07808=1015.159,382.715,-158.366,172.054,51.559,160.401
C07809=1015.170,383.036,-158.420,172.067,51.557,160.402
C07810=1015.182,383.357,-158.473,172.082,51.553,160.404
C07811=1015.193,383.679,-158.527,172.095,51.551,160.406
C07812=1015.205,384.000,-158.580,172.109,51.547,160.408
C07813=1015.214,384.247,-158.621,172.119,51.546,160.409
C07814=1015.223,384.494,-158.662,172.130,51.543,160.410
C07815=1015.232,384.740,-158.704,172.140,51.540,160.412
C07816=1015.241,384.987,-158.746,172.151,51.539,160.413
C07817=1015.249,385.232,-158.787,172.161,51.536,160.415
C07818=1015.258,385.479,-158.828,172.172,51.535,160.416
C07819=1015.267,385.726,-158.870,172.182,51.532,160.417
C07820=1015.276,385.972,-158.912,172.194,51.530,160.419
C07821=1015.284,386.218,-158.953,172.203,51.528,160.420
C07822=1015.293,386.465,-158.995,172.215,51.526,160.422
C07823=1015.303,386.711,-159.036,172.225,51.524,160.423
C07824=1015.312,386.957,-159.078,172.236,51.522,160.425
C07825=1015.321,387.203,-159.120,172.247,51.520,160.426
C07826=1015.330,387.450,-159.161,172.258,51.517,160.428
C07827=1015.339,387.696,-159.203,172.268,51.516,160.429
C07828=1015.347,387.942,-159.246,172.279,51.514,160.431
C07829=1015.356,388.189,-159.288,172.290,51.512,160.432
C07830=1015.365,388.435,-159.329,172.301,51.509,160.434
C07831=1015.374,388.681,-159.371,172.311,51.508,160.435
C07832=1015.383,388.927,-159.414,172.322,51.506,160.437
C07833=1015.392,389.173,-159.455,172.334,51.504,160.438
C07834=1015.401,389.419,-159.498,172.345,51.502,160.440
C07835=1015.410,389.665,-159.539,172.355,51.500,160.441
C07836=1015.420,389.911,-159.582,172.366,51.498,160.443
C07837=1015.428,390.159,-159.625,172.377,51.497,160.444
C07838=1015.438,390.404,-159.667,172.389,51.495,160.446
C07839=1015.447,390.651,-159.709,172.400,51.493,160.448
C07840=1015.456,390.896,-159.751,172.411,51.491,160.449
C07841=1015.466,391.143,-159.794,172.423,51.489,160.451
C07842=1015.475,391.389,-159.836,172.433,51.488,160.452
C07843=1015.484,391.635,-159.878,172.444,51.486,160.454
C07844=1015.494,391.881,-159.921,172.455,51.484,160.456
C07845=1015.502,392.128,-159.964,172.466,51.482,160.457
C07846=1015.511,392.374,-160.006,172.478,51.480,160.459
C07847=1015.521,392.620,-160.048,172.489,51.479,160.460
C07848=1015.530,392.866,-160.091,172.501,51.477,160.462
C07849=1015.539,393.112,-160.134,172.512,51.475,160.464
C07850=1015.549,393.358,-160.177,172.523,51.473,160.465
C07851=1015.557,393.604,-160.220,172.535,51.472,160.467
C07852=1015.567,393.850,-160.263,172.546,51.470,160.469
C07853=1015.576,394.096,-160.306,172.558,51.469,160.470
C07854=1015.586,394.343,-160.348,172.569,51.467,160.472
C07855=1015.595,394.589,-160.391,172.581,51.465,160.474
C07856=1015.605,394.835,-160.435,172.592,51.464,160.476
C07857=1015.614,395.080,-160.477,172.604,51.462,160.477
C07858=1015.623,395.327,-160.521,172.615,51.460,160.479
C07859=1015.633,395.573,-160.564,172.627,51.459,160.481
C07860=1015.643,395.819,-160.607,172.638,51.458,160.483
C07861=1015.653,396.065,-160.650,172.650,51.456,160.484
C07862=1015.662,396.311,-160.694,172.661,51.454,160.486
C07863=1015.671,396.557,-160.736,172.674,51.453,160.488
C07864=1015.681,396.803,-160.780,172.685,51.451,160.490
C07865=1015.691,397.049,-160.824,172.697,51.450,160.491
C07866=1015.700,397.295,-160.866,172.708,51.449,160.493
C07867=1015.709,397.541,-160.910,172.720,51.447,160.495
C07868=1015.720,397.787,-160.954,172.732,51.446,160.497
C07869=1015.736,398.202,-161.027,172.752,51.443,160.500
C07870=1015.751,398.617,-161.101,172.772,51.441,160.503
C07871=1015.398,396.589,-161.087,172.658,51.516,160.502
C07872=1015.388,396.343,-161.044,172.647,51.518,160.501
C07873=1015.379,396.096,-161.000,172.635,51.520,160.499
C07874=1015.369,395.851,-160.957,172.622,51.522,160.497
C07875=1015.359,395.605,-160.914,172.611,51.523,160.495
C07876=1015.349,395.359,-160.871,172.600,51.525,160.494
C07877=1015.341,395.113,-160.828,172.588,51.526,160.492
C07878=1015.331,394.867,-160.785,172.577,51.528,160.490
C07879=1015.322,394.621,-160.743,172.565,51.530,160.488
C07880=1015.312,394.375,-160.699,172.554,51.531,160.487
C07881=1015.303,394.129,-160.656,172.542,51.533,160.485
C07882=1015.293,393.883,-160.613,172.531,51.534,160.483
C07883=1015.284,393.637,-160.571,172.519,51.537,160.482
C07884=1015.275,393.390,-160.528,172.507,51.539,160.480
C07885=1015.266,393.144,-160.485,172.496,51.540,160.478
C07886=1015.256,392.899,-160.443,172.484,51.542,160.477
C07887=1015.247,392.652,-160.399,172.473,51.544,160.475
C07888=1015.238,392.406,-160.357,172.462,51.545,160.473
C07889=1015.229,392.160,-160.314,172.450,51.547,160.472
C07890=1015.219,391.914,-160.272,172.439,51.549,160.470
C07891=1015.211,391.667,-160.229,172.429,51.550,160.468
C07892=1015.201,391.421,-160.187,172.417,51.552,160.467
C07893=1015.192,391.175,-160.144,172.406,51.554,160.465
C07894=1015.183,390.929,-160.102,172.395,51.556,160.464
C07895=1015.173,390.683,-160.060,172.384,51.558,160.462
C07896=1015.164,390.437,-160.017,172.373,51.560,160.461
C07897=1015.155,390.190,-159.975,172.361,51.562,160.459
C07898=1015.145,389.944,-159.933,172.350,51.564,160.457
C07899=1015.137,389.698,-159.891,172.339,51.566,160.456
C07900=1015.128,389.452,-159.848,172.328,51.568,160.454
C07901=1015.119,389.206,-159.806,172.317,51.570,160.453
C07902=1015.110,388.959,-159.765,172.307,51.572,160.451
C07903=1015.101,388.713,-159.722,172.296,51.574,160.450
C07904=1015.092,388.467,-159.681,172.284,51.576,160.448
C07905=1015.083,388.221,-159.639,172.273,51.578,160.447
C07906=1015.074,387.974,-159.597,172.262,51.580,160.445
C07907=1015.065,387.729,-159.555,172.252,51.582,160.444
C07908=1015.056,387.482,-159.513,172.241,51.584,160.442
C07909=1015.047,387.236,-159.471,172.230,51.586,160.441
C07910=1015.038,386.989,-159.430,172.219,51.589,160.439
C07911=1015.029,386.743,-159.388,172.209,51.590,160.438
C07912=1015.020,386.497,-159.346,172.198,51.593,160.436
C07913=1015.011,386.250,-159.304,172.187,51.595,160.435
C07914=1015.002,386.004,-159.263,172.176,51.598,160.434
C07915=1014.993,385.758,-159.221,172.166,51.599,160.432
C07916=1014.985,385.511,-159.180,172.155,51.602,160.431
C07917=1014.976,385.265,-159.139,172.144,51.604,160.429
C07918=1014.968,385.019,-159.097,172.134,51.606,160.428
C07919=1014.959,384.772,-159.055,172.123,51.608,160.426
C07920=1014.950,384.525,-159.014,172.112,51.611,160.425
C07921=1014.941,384.279,-158.973,172.102,51.613,160.424
C07922=1014.932,384.033,-158.932,172.091,51.615,160.422
C07923=1014.923,383.787,-158.891,172.081,51.618,160.421
C07924=1014.915,383.537,-158.849,172.071,51.620,160.420
C07925=1014.906,383.289,-158.809,172.060,51.622,160.418
C07926=1014.897,383.040,-158.766,172.049,51.625,160.417
C07927=1014.888,382.792,-158.726,172.039,51.627,160.415
C07928=1014.879,382.545,-158.685,172.028,51.629,160.414
C07929=1014.871,382.299,-158.643,172.018,51.631,160.413
C07930=1014.862,382.052,-158.602,172.008,51.634,160.411
C07931=1014.853,381.806,-158.562,171.997,51.636,160.410
C07932=1014.845,381.559,-158.521,171.987,51.639,160.409
C07933=1014.836,381.312,-158.480,171.977,51.642,160.408
C07934=1014.827,381.067,-158.439,171.967,51.644,160.406
C07935=1014.818,380.820,-158.398,171.956,51.646,160.405
C07936=1014.810,380.574,-158.358,171.946,51.649,160.404
C07937=1014.801,380.327,-158.317,171.935,51.651,160.402
C07938=1014.793,380.081,-158.277,171.926,51.653,160.401
C07939=1014.784,379.834,-158.236,171.915,51.657,160.400
C07940=1014.776,379.587,-158.195,171.905,51.659,160.399
C07941=1014.767,379.341,-158.155,171.895,51.661,160.397
C07942=1014.759,379.094,-158.114,171.885,51.664,160.396
C07943=1014.751,378.848,-158.073,171.875,51.666,160.395
C07944=1014.742,378.601,-158.034,171.865,51.669,160.394
C07945=1014.734,378.355,-157.993,171.855,51.672,160.393
C07946=1014.726,378.108,-157.952,171.844,51.674,160.391
C07947=1014.717,377.861,-157.911,171.835,51.677,160.390
C07948=1014.709,377.615,-157.872,171.825,51.679,160.389
C07949=1014.701,377.368,-157.831,171.815,51.682,160.388
C07950=1014.693,377.122,-157.791,171.805,51.684,160.386
C07951=1014.684,376.875,-157.751,171.796,51.687,160.385
C07952=1014.676,376.629,-157.711,171.785,51.690,160.384
C07953=1014.667,376.382,-157.670,171.775,51.693,160.383
C07954=1014.660,376.135,-157.630,171.766,51.695,160.382
C07955=1014.651,375.889,-157.590,171.755,51.698,160.381
C07956=1014.643,375.643,-157.550,171.746,51.701,160.380
C07957=1014.635,375.396,-157.509,171.736,51.704,160.378
C07958=1014.626,375.149,-157.470,171.726,51.706,160.377
C07959=1014.618,374.902,-157.430,171.716,51.709,160.376
C07960=1014.610,374.655,-157.390,171.707,51.712,160.375
C07961=1014.602,374.409,-157.351,171.697,51.715,160.374
C07962=1014.594,374.163,-157.310,171.687,51.718,160.373
C07963=1014.585,373.916,-157.271,171.678,51.720,160.372
C07964=1014.577,373.669,-157.232,171.668,51.723,160.371
C07965=1014.569,373.422,-157.192,171.658,51.726,160.370
C07966=1014.560,373.176,-157.153,171.649,51.729,160.368
C07967=1014.553,372.929,-157.113,171.639,51.732,160.367
C07968=1014.544,372.682,-157.073,171.630,51.735,160.366
C07969=1014.536,372.436,-157.034,171.619,51.738,160.365
C07970=1014.528,372.189,-156.994,171.610,51.741,160.364
C07971=1014.520,371.942,-156.955,171.601,51.744,160.363
C07972=1014.511,371.695,-156.916,171.591,51.746,160.362
C07973=1014.504,371.448,-156.876,171.581,51.749,160.361
C07974=1014.495,371.202,-156.837,171.572,51.753,160.360
C07975=1014.488,370.955,-156.797,171.562,51.756,160.359
C07976=1014.479,370.708,-156.758,171.553,51.758,160.358
C07977=1014.472,370.462,-156.719,171.544,51.761,160.357
C07978=1014.464,370.215,-156.680,171.535,51.765,160.356
C07979=1014.455,369.968,-156.640,171.525,51.767,160.355
C07980=1014.447,369.721,-156.602,171.515,51.771,160.354
C07981=1014.440,369.475,-156.562,171.506,51.774,160.353
C07982=1014.432,369.227,-156.523,171.497,51.777,160.352
C07983=1014.424,368.980,-156.483,171.487,51.780,160.351
C07984=1014.415,368.680,-156.436,171.476,51.784,160.350
C07985=1014.405,368.378,-156.389,171.465,51.787,160.349
C07986=1014.396,368.077,-156.341,171.453,51.791,160.347
C07987=1014.386,367.776,-156.293,171.442,51.795,160.346
C07988=1014.378,367.530,-156.254,171.433,51.798,160.345
C07989=1014.371,367.283,-156.215,171.424,51.801,160.344
C07990=1014.362,367.035,-156.177,171.415,51.804,160.343
C07991=1014.355,366.789,-156.138,171.405,51.808,160.342
C07992=1014.346,366.542,-156.099,171.396,51.811,160.341
C07993=1014.339,366.296,-156.061,171.387,51.815,160.341
C07994=1014.331,366.049,-156.022,171.377,51.817,160.340
C07995=1014.323,365.801,-155.984,171.368,51.821,160.339
C07996=1014.315,365.555,-155.945,171.359,51.824,160.338
C07997=1014.307,365.308,-155.907,171.350,51.828,160.337
C07998=1014.299,365.061,-155.869,171.341,51.831,160.336
C07999=1014.291,364.814,-155.830,171.332,51.834,160.335
C08000=1014.284,364.567,-155.791,171.323,51.837,160.334
C08001=1014.276,364.320,-155.752,171.314,51.841,160.333
C08002=1014.269,364.073,-155.715,171.305,51.844,160.333
C08003=1014.261,363.826,-155.677,171.296,51.848,160.332
C08004=1014.253,363.579,-155.638,171.287,51.851,160.331
C08005=1014.246,363.332,-155.600,171.278,51.854,160.330
C08006=1014.238,363.085,-155.561,171.269,51.858,160.329
C08007=1014.230,362.838,-155.524,171.260,51.861,160.328
C08008=1014.223,362.592,-155.485,171.251,51.865,160.327
C08009=1014.215,362.344,-155.447,171.242,51.868,160.327
C08010=1014.207,362.097,-155.409,171.233,51.872,160.326
C08011=1014.200,361.851,-155.371,171.224,51.875,160.325
C08012=1014.192,361.603,-155.333,171.215,51.878,160.324
C08013=1014.184,361.356,-155.295,171.208,51.882,160.324
C08014=1014.177,361.110,-155.257,171.199,51.885,160.323
C08015=1014.170,360.863,-155.219,171.190,51.889,160.322
C08016=1014.161,360.615,-155.181,171.181,51.892,160.321
C08017=1014.154,360.368,-155.143,171.172,51.896,160.320
C08018=1014.147,360.121,-155.106,171.163,51.900,160.319
C08019=1014.139,359.875,-155.067,171.154,51.903,160.319
C08020=1014.132,359.628,-155.030,171.145,51.907,160.318
C08021=1014.125,359.381,-154.992,171.137,51.911,160.317
C08022=1014.117,359.134,-154.954,171.129,51.914,160.316
C08023=1014.110,358.886,-154.916,171.120,51.917,160.316
C08024=1014.102,358.640,-154.878,171.111,51.921,160.315
C08025=1014.095,358.392,-154.840,171.102,51.925,160.314
C08026=1014.088,358.145,-154.803,171.094,51.929,160.313
C08027=1014.080,357.898,-154.765,171.085,51.932,160.313
C08028=1014.073,357.651,-154.728,171.076,51.936,160.312
C08029=1014.065,357.404,-154.691,171.068,51.939,160.311
C08030=1014.058,357.157,-154.653,171.060,51.943,160.311
C08031=1014.051,356.910,-154.616,171.051,51.947,160.310
C08032=1014.043,356.663,-154.578,171.042,51.951,160.309
C08033=1014.035,356.416,-154.541,171.034,51.955,160.308
C08034=1014.028,356.169,-154.504,171.025,51.958,160.308
C08035=1014.021,355.922,-154.466,171.017,51.962,160.307
C08036=1014.014,355.674,-154.429,171.009,51.966,160.306
C08037=1014.006,355.427,-154.392,171.000,51.969,160.305
C08038=1013.999,355.180,-154.355,170.991,51.973,160.305
C08039=1013.991,354.933,-154.317,170.982,51.977,160.304
C08040=1013.984,354.685,-154.281,170.975,51.981,160.304
C08041=1013.977,354.439,-154.244,170.966,51.985,160.303
C08042=1013.970,354.192,-154.207,170.957,51.989,160.302
C08043=1013.963,353.944,-154.170,170.949,51.993,160.302
C08044=1013.954,353.651,-154.126,170.939,51.997,160.301
C08045=1013.946,353.357,-154.082,170.929,52.002,160.300
C08046=1013.936,353.063,-154.038,170.919,52.006,160.299
C08047=1013.928,352.770,-153.994,170.910,52.011,160.298
C08048=1013.921,352.523,-153.958,170.901,52.015,160.298
C08049=1013.913,352.276,-153.921,170.893,52.020,160.297
C08050=1013.906,352.029,-153.884,170.884,52.024,160.297
C08051=1013.898,351.782,-153.847,170.877,52.027,160.296
C08052=1013.892,351.535,-153.810,170.868,52.031,160.296
C08053=1013.884,351.287,-153.774,170.860,52.035,160.295
C08054=1013.877,351.040,-153.737,170.851,52.040,160.294
C08055=1013.869,350.793,-153.701,170.843,52.043,160.294
C08056=1013.863,350.546,-153.664,170.835,52.047,160.293
C08057=1013.855,350.298,-153.628,170.826,52.051,160.292
C08058=1013.849,350.051,-153.591,170.818,52.056,160.292
C08059=1013.841,349.804,-153.554,170.811,52.060,160.292
C08060=1013.834,349.557,-153.518,170.802,52.064,160.291
C08061=1013.827,349.310,-153.482,170.794,52.068,160.290
C08062=1013.820,349.062,-153.445,170.786,52.072,160.290
C08063=1013.814,348.815,-153.409,170.778,52.076,160.289
C08064=1013.806,348.568,-153.372,170.769,52.080,160.289
C08065=1013.800,348.321,-153.336,170.762,52.084,160.288
C08066=1013.792,348.073,-153.300,170.754,52.089,160.288
C08067=1013.785,347.825,-153.263,170.745,52.093,160.287
C08068=1013.778,347.579,-153.227,170.738,52.097,160.287
C08069=1013.772,347.332,-153.191,170.729,52.101,160.286
C08070=1013.764,347.084,-153.154,170.721,52.105,160.285
C08071=1013.757,346.837,-153.119,170.714,52.110,160.285
C08072=1013.750,346.589,-153.082,170.705,52.114,160.284
C08073=1013.743,346.342,-153.047,170.697,52.118,160.284
C08074=1013.736,346.094,-153.010,170.689,52.122,160.283
C08075=1013.729,345.848,-152.974,170.681,52.127,160.283
C08076=1013.723,345.600,-152.939,170.673,52.132,160.283
C08077=1013.715,345.353,-152.903,170.666,52.135,160.282
C08078=1013.709,345.106,-152.866,170.657,52.140,160.282
C08079=1013.701,344.858,-152.831,170.649,52.144,160.281
C08080=1013.694,344.611,-152.795,170.642,52.148,160.281
C08081=1013.688,344.363,-152.759,170.634,52.153,160.280
C08082=1013.680,344.116,-152.723,170.625,52.158,160.280
C08083=1013.674,343.869,-152.688,170.618,52.161,160.279
C08084=1013.667,343.622,-152.652,170.610,52.166,160.279
C08085=1013.661,343.374,-152.616,170.602,52.171,160.278
C08086=1013.653,343.127,-152.580,170.595,52.175,160.278
C08087=1013.646,342.879,-152.545,170.586,52.179,160.277
C08088=1013.639,342.632,-152.510,170.579,52.184,160.277
C08089=1013.633,342.385,-152.473,170.571,52.188,160.277
C08090=1013.626,342.137,-152.438,170.563,52.193,160.276
C08091=1013.619,341.890,-152.403,170.555,52.197,160.276
C08092=1013.612,341.643,-152.367,170.547,52.202,160.275
C08093=1013.605,341.395,-152.332,170.540,52.207,160.275
C08094=1013.599,341.148,-152.296,170.532,52.211,160.274
C08095=1013.592,340.900,-152.260,170.523,52.215,160.274
C08096=1013.585,340.652,-152.225,170.516,52.220,160.274
C08097=1013.578,340.406,-152.189,170.508,52.224,160.273
C08098=1013.571,340.158,-152.154,170.501,52.229,160.273
C08099=1013.565,339.911,-152.118,170.493,52.233,160.272
C08100=1013.558,339.663,-152.083,170.486,52.238,160.272
C08101=1013.551,339.416,-152.048,170.478,52.243,160.272
C08102=1013.545,339.168,-152.013,170.470,52.248,160.271
C08103=1013.538,338.921,-151.978,170.463,52.252,160.271
C08104=1013.530,338.625,-151.935,170.454,52.257,160.270
C08105=1013.522,338.329,-151.894,170.444,52.264,160.270
C08106=1013.514,338.032,-151.852,170.435,52.269,160.270
C08107=1013.506,337.737,-151.810,170.426,52.274,160.269
C08108=1013.499,337.489,-151.775,170.418,52.279,160.269
C08109=1013.492,337.241,-151.740,170.411,52.284,160.269
C08110=1013.486,336.994,-151.705,170.403,52.289,160.268
C08111=1013.479,336.747,-151.670,170.396,52.293,160.268
C08112=1013.472,336.499,-151.636,170.388,52.299,160.268
C08113=1013.466,336.251,-151.601,170.380,52.303,160.267
C08114=1013.459,336.004,-151.565,170.373,52.308,160.267
C08115=1013.452,335.756,-151.531,170.365,52.313,160.267
C08116=1013.445,335.510,-151.497,170.358,52.317,160.266
C08117=1013.439,335.262,-151.462,170.350,52.322,160.266
C08118=1013.432,335.014,-151.427,170.343,52.327,160.266
C08119=1013.425,334.767,-151.392,170.335,52.332,160.265
C08120=1013.419,334.519,-151.358,170.329,52.337,160.265
C08121=1013.412,334.271,-151.323,170.321,52.342,160.265
C08122=1013.406,334.024,-151.288,170.314,52.347,160.265
C08123=1013.400,333.777,-151.253,170.306,52.351,160.264
C08124=1013.393,333.529,-151.219,170.299,52.356,160.264
C08125=1013.387,333.281,-151.185,170.291,52.361,160.264
C08126=1013.380,333.034,-151.150,170.283,52.367,160.263
C08127=1013.374,332.786,-151.115,170.276,52.371,160.263
C08128=1013.366,332.539,-151.081,170.268,52.376,160.263
C08129=1013.360,332.291,-151.046,170.262,52.381,160.263
C08130=1013.354,332.044,-151.012,170.254,52.386,160.262
C08131=1013.347,331.797,-150.977,170.247,52.391,160.262
C08132=1013.341,331.549,-150.943,170.239,52.397,160.262
C08133=1013.334,331.302,-150.909,170.232,52.401,160.262
C08134=1013.328,331.054,-150.875,170.224,52.406,160.261
C08135=1013.321,330.806,-150.840,170.218,52.411,160.261
C08136=1013.315,330.559,-150.807,170.210,52.417,160.261
C08137=1013.308,330.311,-150.773,170.203,52.422,160.261
C08138=1013.302,330.063,-150.738,170.195,52.427,160.260
C08139=1013.295,329.816,-150.705,170.188,52.432,160.260
C08140=1013.289,329.568,-150.670,170.181,52.437,160.260
C08141=1013.283,329.320,-150.636,170.174,52.442,160.260
C08142=1013.276,329.073,-150.602,170.166,52.447,160.260
C08143=1013.270,328.825,-150.568,170.160,52.452,160.260
C08144=1013.263,328.577,-150.534,170.152,52.458,160.259
C08145=1013.256,328.330,-150.500,170.145,52.463,160.259
C08146=1013.250,328.083,-150.466,170.138,52.468,160.259
C08147=1013.243,327.835,-150.432,170.130,52.473,160.259
C08148=1013.238,327.587,-150.399,170.123,52.478,160.258
C08149=1013.232,327.340,-150.365,170.116,52.483,160.258
C08150=1013.225,327.092,-150.331,170.108,52.488,160.258
C08151=1013.219,326.845,-150.297,170.102,52.494,160.258
C08152=1013.212,326.597,-150.263,170.094,52.500,160.258
C08153=1013.206,326.349,-150.230,170.088,52.505,160.258
C08154=1013.199,326.101,-150.195,170.080,52.510,160.257
C08155=1013.194,325.854,-150.161,170.073,52.515,160.257
C08156=1013.187,325.606,-150.129,170.067,52.520,160.257
C08157=1013.180,325.359,-150.095,170.059,52.526,160.257
C08158=1013.175,325.111,-150.061,170.051,52.531,160.257
C08159=1013.168,324.864,-150.028,170.045,52.537,160.257
C08160=1013.161,324.615,-149.995,170.037,52.542,160.257
C08161=1013.154,324.368,-149.961,170.031,52.547,160.256
C08162=1013.148,324.121,-149.929,170.023,52.553,160.256
C08163=1013.142,323.872,-149.895,170.017,52.558,160.256
C08164=1013.134,323.572,-149.855,170.008,52.565,160.256
C08165=1013.126,323.272,-149.814,169.999,52.572,160.256
C08166=1013.118,322.971,-149.774,169.991,52.578,160.256
C08167=1013.111,322.671,-149.734,169.983,52.584,160.256
C08168=1013.104,322.423,-149.701,169.975,52.591,160.256
C08169=1013.098,322.176,-149.668,169.969,52.596,160.256
C08170=1013.091,321.927,-149.635,169.961,52.601,160.255
C08171=1013.085,321.680,-149.601,169.955,52.607,160.255
C08172=1013.079,321.432,-149.568,169.947,52.612,160.255
C08173=1013.073,321.185,-149.536,169.941,52.618,160.255
C08174=1013.066,320.937,-149.503,169.933,52.623,160.255
C08175=1013.060,320.689,-149.470,169.927,52.629,160.255
C08176=1013.053,320.441,-149.437,169.919,52.634,160.255
C08177=1013.048,320.193,-149.404,169.913,52.640,160.255
C08178=1013.041,319.946,-149.371,169.906,52.646,160.255
C08179=1013.035,319.698,-149.338,169.899,52.651,160.255
C08180=1013.029,319.451,-149.306,169.892,52.657,160.255
C08181=1013.023,319.203,-149.273,169.885,52.663,160.255
C08182=1013.017,318.955,-149.239,169.878,52.669,160.255
C08183=1013.010,318.707,-149.206,169.872,52.674,160.255
C08184=1013.004,318.459,-149.174,169.864,52.680,160.255
C08185=1012.998,318.212,-149.141,169.858,52.685,160.255
C08186=1012.991,317.964,-149.108,169.850,52.692,160.255
C08187=1012.986,317.716,-149.075,169.844,52.697,160.254
C08188=1012.979,317.469,-149.042,169.837,52.703,160.254
C08189=1012.973,317.220,-149.010,169.830,52.708,160.255
C08190=1012.967,316.973,-148.977,169.824,52.714,160.255
C08191=1012.961,316.725,-148.945,169.816,52.720,160.254
C08192=1012.955,316.478,-148.912,169.810,52.725,160.254
C08193=1012.949,316.230,-148.878,169.803,52.731,160.254
C08194=1012.944,315.982,-148.847,169.797,52.737,160.255
C08195=1012.937,315.735,-148.814,169.789,52.743,160.254
C08196=1012.931,315.487,-148.781,169.783,52.748,160.254
C08197=1012.925,315.239,-148.749,169.775,52.755,160.254
C08198=1012.919,314.991,-148.716,169.769,52.760,160.254
C08199=1012.913,314.743,-148.683,169.763,52.766,160.254
C08200=1012.907,314.495,-148.651,169.756,52.772,160.254
C08201=1012.901,314.247,-148.618,169.750,52.778,160.255
C08202=1012.895,314.001,-148.586,169.742,52.784,160.254
C08203=1012.889,313.752,-148.554,169.736,52.790,160.255
C08204=1012.884,313.504,-148.521,169.729,52.796,160.255
C08205=1012.878,313.256,-148.489,169.723,52.802,160.255
C08206=1012.871,313.009,-148.456,169.715,52.808,160.255
C08207=1012.866,312.761,-148.424,169.709,52.813,160.255
C08208=1012.860,312.514,-148.392,169.703,52.819,160.255
C08209=1012.854,312.265,-148.359,169.696,52.825,160.255
C08210=1012.848,312.017,-148.326,169.689,52.831,160.255
C08211=1012.843,311.770,-148.294,169.682,52.837,160.255
C08212=1012.836,311.522,-148.262,169.676,52.843,160.255
C08213=1012.830,311.274,-148.230,169.670,52.849,160.255
C08214=1012.825,311.027,-148.197,169.662,52.855,160.255
C08215=1012.819,310.779,-148.165,169.656,52.861,160.255
C08216=1012.814,310.530,-148.133,169.649,52.867,160.255
C08217=1012.808,310.284,-148.100,169.643,52.872,160.255
C08218=1012.802,310.035,-148.068,169.637,52.879,160.255
C08219=1012.796,309.787,-148.036,169.630,52.885,160.255
C08220=1012.790,309.540,-148.004,169.624,52.891,160.255
C08221=1012.784,309.292,-147.972,169.616,52.897,160.255
C08222=1012.780,309.044,-147.940,169.610,52.903,160.255
C08223=1012.773,308.796,-147.908,169.603,52.909,160.256
C08224=1012.766,308.501,-147.871,169.595,52.917,160.256
C08225=1012.758,308.207,-147.833,169.588,52.924,160.256
C08226=1012.752,307.911,-147.795,169.580,52.931,160.256
C08227=1012.744,307.616,-147.758,169.573,52.939,160.256
C08228=1012.738,307.369,-147.727,169.565,52.945,160.256
C08229=1012.732,307.121,-147.695,169.560,52.951,160.256
C08230=1012.726,306.873,-147.663,169.552,52.958,160.256
C08231=1012.720,306.625,-147.632,169.547,52.964,160.257
C08232=1012.714,306.377,-147.601,169.539,52.970,160.257
C08233=1012.708,306.130,-147.569,169.534,52.977,160.257
C08234=1012.702,305.882,-147.538,169.526,52.983,160.257
C08235=1012.697,305.634,-147.507,169.521,52.989,160.257
C08236=1012.690,305.386,-147.475,169.514,52.995,160.257
C08237=1012.684,305.138,-147.444,169.508,53.002,160.257
C08238=1012.678,304.890,-147.413,169.501,53.008,160.258
C08239=1012.673,304.642,-147.381,169.495,53.014,160.258
C08240=1012.666,304.394,-147.350,169.489,53.021,160.258
C08241=1012.661,304.146,-147.319,169.482,53.027,160.258
C08242=1012.655,303.899,-147.288,169.476,53.033,160.258
C08243=1012.649,303.650,-147.257,169.469,53.040,160.258
C08244=1012.643,303.403,-147.226,169.463,53.046,160.259
C08245=1012.637,303.154,-147.194,169.456,53.053,160.259
C08246=1012.631,302.907,-147.163,169.450,53.059,160.259
C08247=1012.626,302.659,-147.132,169.443,53.065,160.259
C08248=1012.620,302.410,-147.100,169.437,53.072,160.259
C08249=1012.614,302.163,-147.070,169.431,53.079,160.259
C08250=1012.608,301.914,-147.038,169.425,53.085,160.260
C08251=1012.602,301.667,-147.007,169.418,53.092,160.260
C08252=1012.597,301.419,-146.976,169.412,53.098,160.260
C08253=1012.591,301.171,-146.945,169.405,53.105,160.260
C08254=1012.586,300.922,-146.914,169.399,53.111,160.260
C08255=1012.579,300.675,-146.883,169.392,53.118,160.261
C08256=1012.574,300.427,-146.852,169.387,53.124,160.261
C08257=1012.568,300.179,-146.821,169.379,53.131,160.261
C08258=1012.563,299.931,-146.790,169.374,53.137,160.261
C08259=1012.557,299.683,-146.759,169.367,53.144,160.261
C08260=1012.552,299.435,-146.728,169.361,53.150,160.262
C08261=1012.545,299.187,-146.698,169.354,53.157,160.262
C08262=1012.540,298.939,-146.666,169.349,53.164,160.262
C08263=1012.534,298.691,-146.636,169.343,53.170,160.262
C08264=1012.529,298.443,-146.605,169.336,53.177,160.263
C08265=1012.523,298.195,-146.574,169.330,53.183,160.263
C08266=1012.517,297.947,-146.542,169.324,53.190,160.263
C08267=1012.511,297.699,-146.512,169.318,53.197,160.263
C08268=1012.506,297.451,-146.481,169.311,53.204,160.264
C08269=1012.500,297.203,-146.451,169.305,53.210,160.264
C08270=1012.495,296.955,-146.420,169.299,53.217,160.264
C08271=1012.490,296.707,-146.389,169.293,53.223,160.264
C08272=1012.484,296.459,-146.358,169.286,53.230,160.264
C08273=1012.478,296.211,-146.328,169.280,53.237,160.265
C08274=1012.473,295.963,-146.297,169.274,53.244,160.265
C08275=1012.467,295.715,-146.266,169.268,53.250,160.265
C08276=1012.462,295.467,-146.236,169.262,53.257,160.266
C08277=1012.456,295.219,-146.205,169.255,53.264,160.266
C08278=1012.451,294.971,-146.174,169.250,53.270,160.266
C08279=1012.445,294.723,-146.144,169.243,53.278,160.266
C08280=1012.440,294.475,-146.113,169.238,53.284,160.267
C08281=1012.434,294.227,-146.083,169.231,53.291,160.267
C08282=1012.429,293.979,-146.052,169.225,53.297,160.267
C08283=1012.424,293.731,-146.021,169.218,53.304,160.267
C08284=1012.418,293.454,-145.986,169.212,53.312,160.268
C08285=1012.412,293.177,-145.953,169.205,53.320,160.268
C08286=1012.406,292.901,-145.919,169.198,53.327,160.268
C08287=1012.400,292.624,-145.885,169.192,53.335,160.269
C08288=1012.395,292.376,-145.854,169.185,53.342,160.269
C08289=1012.389,292.128,-145.824,169.180,53.348,160.269
C08290=1012.383,291.880,-145.794,169.173,53.356,160.270
C08291=1012.378,291.632,-145.764,169.168,53.362,160.270
C08292=1012.373,291.384,-145.733,169.161,53.369,160.270
C08293=1012.367,291.135,-145.703,169.156,53.376,160.271
C08294=1012.361,290.887,-145.673,169.149,53.383,160.271
C08295=1012.356,290.639,-145.643,169.144,53.390,160.271
C08296=1012.350,290.391,-145.613,169.137,53.397,160.271
C08297=1012.345,290.143,-145.584,169.132,53.405,160.272
C08298=1012.339,289.895,-145.553,169.125,53.411,160.272
C08299=1012.334,289.647,-145.524,169.119,53.419,160.273
C08300=1012.328,289.399,-145.494,169.113,53.426,160.273
C08301=1012.322,289.151,-145.464,169.107,53.433,160.273
C08302=1012.317,288.902,-145.434,169.101,53.440,160.274
C08303=1012.311,288.655,-145.404,169.095,53.447,160.274
C08304=1012.306,288.407,-145.375,169.089,53.454,160.274
C08305=1012.301,288.158,-145.344,169.083,53.461,160.275
C08306=1012.296,287.910,-145.315,169.077,53.468,160.275
C08307=1012.290,287.662,-145.284,169.070,53.475,160.275
C08308=1012.284,287.413,-145.255,169.065,53.483,160.276
C08309=1012.280,287.166,-145.225,169.059,53.490,160.276
C08310=1012.274,286.917,-145.196,169.053,53.497,160.276
C08311=1012.268,286.669,-145.165,169.047,53.504,160.277
C08312=1012.263,286.421,-145.136,169.041,53.512,160.277
C08313=1012.258,286.173,-145.106,169.035,53.518,160.278
C08314=1012.252,285.925,-145.077,169.029,53.526,160.278
C08315=1012.246,285.677,-145.048,169.023,53.533,160.278
C08316=1012.241,285.429,-145.019,169.017,53.540,160.279
C08317=1012.236,285.180,-144.989,169.011,53.547,160.279
C08318=1012.230,284.932,-144.959,169.005,53.555,160.280
C08319=1012.224,284.684,-144.929,169.000,53.562,160.280
C08320=1012.219,284.436,-144.900,168.994,53.570,160.280
C08321=1012.214,284.188,-144.870,168.988,53.576,160.281
C08322=1012.208,283.939,-144.840,168.982,53.584,160.281
C08323=1012.203,283.692,-144.811,168.975,53.591,160.281
C08324=1012.198,283.443,-144.783,168.970,53.599,160.282
C08325=1012.192,283.195,-144.753,168.964,53.606,160.282
C08326=1012.187,282.947,-144.724,168.959,53.613,160.283
C08327=1012.181,282.699,-144.695,168.952,53.621,160.283
C08328=1012.176,282.451,-144.666,168.946,53.629,160.284
C08329=1012.171,282.202,-144.637,168.941,53.636,160.284
C08330=1012.165,281.953,-144.607,168.935,53.644,160.285
C08331=1012.160,281.706,-144.578,168.929,53.651,160.285
C08332=1012.151,281.335,-144.535,168.920,53.661,160.285
C08333=1012.143,280.964,-144.491,168.911,53.673,160.286
C08334=1012.135,280.594,-144.448,168.902,53.684,160.287
C08335=1012.127,280.222,-144.405,168.893,53.695,160.287
C08336=1011.905,282.016,-144.978,168.907,53.731,160.298
C08337=1011.909,282.229,-145.003,168.911,53.724,160.298
C08338=1011.914,282.440,-145.029,168.916,53.718,160.297
C08339=1011.919,282.652,-145.053,168.922,53.711,160.297
C08340=1011.923,282.864,-145.078,168.927,53.705,160.297
C08341=1011.928,283.076,-145.103,168.931,53.699,160.296
C08342=1011.933,283.289,-145.128,168.937,53.692,160.296
C08343=1011.937,283.501,-145.153,168.942,53.686,160.296
C08344=1011.942,283.712,-145.178,168.947,53.679,160.295
C08345=1011.947,283.960,-145.207,168.953,53.672,160.295
C08346=1011.953,284.209,-145.237,168.959,53.665,160.295
C08347=1011.958,284.457,-145.266,168.965,53.658,160.294
C08348=1011.963,284.705,-145.296,168.971,53.650,160.294
C08349=1011.969,284.953,-145.325,168.976,53.643,160.293
C08350=1011.974,285.201,-145.354,168.982,53.636,160.293
C08351=1011.980,285.449,-145.384,168.989,53.629,160.293
C08352=1011.985,285.698,-145.413,168.994,53.621,160.292
C08353=1011.990,285.946,-145.443,169.001,53.614,160.292
C08354=1011.996,286.194,-145.472,169.006,53.607,160.291
C08355=1012.001,286.442,-145.502,169.013,53.600,160.291
C08356=1012.006,286.690,-145.531,169.019,53.592,160.291
C08357=1012.012,286.939,-145.561,169.024,53.585,160.290
C08358=1012.017,287.187,-145.591,169.031,53.578,160.290
C08359=1012.022,287.434,-145.621,169.036,53.571,160.290
C08360=1012.028,287.683,-145.650,169.042,53.563,160.289
C08361=1012.033,287.931,-145.680,169.048,53.557,160.289
C08362=1012.039,288.180,-145.709,169.054,53.549,160.289
C08363=1012.045,288.427,-145.740,169.060,53.542,160.288
C08364=1012.050,288.675,-145.769,169.066,53.535,160.288
C08365=1012.055,288.924,-145.799,169.073,53.528,160.288
C08366=1012.061,289.172,-145.828,169.078,53.521,160.287
C08367=1012.066,289.420,-145.859,169.085,53.513,160.287
C08368=1012.072,289.668,-145.888,169.090,53.507,160.287
C08369=1012.077,289.916,-145.918,169.096,53.499,160.286
C08370=1012.083,290.164,-145.948,169.102,53.492,160.286
C08371=1012.088,290.412,-145.978,169.108,53.485,160.286
C08372=1012.093,290.660,-146.009,169.115,53.478,160.285
C08373=1012.099,290.909,-146.038,169.121,53.471,160.285
C08374=1012.105,291.157,-146.069,169.127,53.464,160.285
C08375=1012.110,291.405,-146.098,169.133,53.457,160.284
C08376=1012.116,291.653,-146.129,169.139,53.450,160.284
C08377=1012.121,291.901,-146.158,169.145,53.443,160.284
C08378=1012.127,292.148,-146.188,169.152,53.436,160.284
C08379=1012.132,292.397,-146.219,169.157,53.429,160.283
C08380=1012.137,292.645,-146.249,169.164,53.422,160.283
C08381=1012.144,292.924,-146.284,169.170,53.415,160.282
C08382=1012.149,293.202,-146.317,169.177,53.407,160.282
C08383=1012.155,293.482,-146.352,169.184,53.399,160.282
C08384=1012.161,293.761,-146.386,169.191,53.391,160.281
C08385=1012.166,294.009,-146.417,169.198,53.384,160.281
C08386=1012.172,294.257,-146.447,169.203,53.378,160.281
C08387=1012.177,294.505,-146.478,169.210,53.371,160.281
C08388=1012.182,294.753,-146.509,169.216,53.364,160.281
C08389=1012.188,295.001,-146.539,169.223,53.358,160.280
C08390=1012.193,295.249,-146.570,169.228,53.350,160.280
C08391=1012.199,295.497,-146.600,169.234,53.344,160.280
C08392=1012.204,295.745,-146.631,169.240,53.337,160.279
C08393=1012.210,295.993,-146.662,169.246,53.331,160.279
C08394=1012.215,296.241,-146.693,169.253,53.324,160.279
C08395=1012.221,296.489,-146.723,169.259,53.317,160.279
C08396=1012.226,296.737,-146.754,169.265,53.310,160.279
C08397=1012.232,296.985,-146.784,169.271,53.304,160.278
C08398=1012.237,297.233,-146.815,169.278,53.297,160.278
C08399=1012.243,297.482,-146.846,169.284,53.290,160.278
C08400=1012.248,297.730,-146.877,169.290,53.284,160.278
C08401=1012.254,297.978,-146.907,169.296,53.277,160.277
C08402=1012.259,298.226,-146.938,169.303,53.270,160.277
C08403=1012.265,298.474,-146.969,169.309,53.264,160.277
C08404=1012.271,298.721,-147.000,169.315,53.257,160.277
C08405=1012.276,298.969,-147.031,169.322,53.250,160.277
C08406=1012.282,299.218,-147.062,169.328,53.243,160.276
C08407=1012.288,299.466,-147.092,169.335,53.237,160.276
C08408=1012.293,299.714,-147.123,169.340,53.230,160.276
C08409=1012.299,299.961,-147.154,169.347,53.223,160.276
C08410=1012.304,300.209,-147.185,169.353,53.217,160.275
C08411=1012.311,300.458,-147.216,169.360,53.210,160.275
C08412=1012.316,300.706,-147.247,169.366,53.204,160.275
C08413=1012.322,300.953,-147.278,169.373,53.197,160.275
C08414=1012.327,301.201,-147.309,169.378,53.191,160.275
C08415=1012.333,301.449,-147.340,169.385,53.184,160.274
C08416=1012.339,301.697,-147.371,169.391,53.177,160.274
C08417=1012.344,301.945,-147.402,169.398,53.171,160.274
C08418=1012.350,302.193,-147.434,169.404,53.165,160.274
C08419=1012.356,302.441,-147.465,169.410,53.158,160.274
C08420=1012.361,302.689,-147.495,169.416,53.152,160.273
C08421=1012.367,302.937,-147.527,169.423,53.145,160.273
C08422=1012.373,303.185,-147.557,169.429,53.139,160.273
C08423=1012.379,303.433,-147.589,169.436,53.132,160.273
C08424=1012.385,303.681,-147.620,169.442,53.126,160.273
C08425=1012.390,303.929,-147.651,169.449,53.119,160.273
C08426=1012.397,304.177,-147.682,169.455,53.113,160.272
C08427=1012.402,304.425,-147.714,169.461,53.106,160.272
C08428=1012.408,304.672,-147.744,169.468,53.100,160.272
C08429=1012.414,304.921,-147.776,169.474,53.093,160.272
C08430=1012.420,305.168,-147.807,169.481,53.088,160.272
C08431=1012.426,305.417,-147.838,169.487,53.081,160.272
C08432=1012.432,305.664,-147.870,169.494,53.074,160.272
C08433=1012.438,305.912,-147.902,169.500,53.068,160.271
C08434=1012.444,306.160,-147.932,169.507,53.061,160.271
C08435=1012.450,306.408,-147.964,169.513,53.056,160.271
C08436=1012.456,306.655,-147.995,169.520,53.049,160.271
C08437=1012.461,306.904,-148.026,169.526,53.043,160.271
C08438=1012.468,307.151,-148.057,169.533,53.036,160.271
C08439=1012.474,307.400,-148.089,169.539,53.030,160.271
C08440=1012.480,307.647,-148.120,169.546,53.024,160.271
C08441=1012.487,307.945,-148.158,169.554,53.016,160.270
C08442=1012.494,308.242,-148.196,169.561,53.008,160.270
C08443=1012.501,308.538,-148.234,169.570,53.001,160.270
C08444=1012.509,308.836,-148.272,169.578,52.994,160.270
C08445=1012.515,309.084,-148.304,169.584,52.988,160.270
C08446=1012.520,309.331,-148.335,169.591,52.981,160.270
C08447=1012.526,309.580,-148.367,169.597,52.975,160.270
C08448=1012.531,309.828,-148.400,169.604,52.969,160.270
C08449=1012.537,310.075,-148.432,169.610,52.963,160.270
C08450=1012.542,310.323,-148.464,169.618,52.957,160.270
C08451=1012.548,310.571,-148.496,169.623,52.951,160.269
C08452=1012.555,310.818,-148.529,169.630,52.945,160.269
C08453=1012.560,311.066,-148.560,169.637,52.939,160.269
C08454=1012.566,311.314,-148.593,169.643,52.933,160.269
C08455=1012.571,311.562,-148.626,169.650,52.927,160.269
C08456=1012.577,311.810,-148.657,169.657,52.921,160.269
C08457=1012.583,312.058,-148.690,169.664,52.915,160.269
C08458=1012.589,312.305,-148.722,169.670,52.909,160.269
C08459=1012.595,312.553,-148.754,169.677,52.903,160.269
C08460=1012.601,312.800,-148.787,169.684,52.897,160.269
C08461=1012.606,313.049,-148.819,169.690,52.891,160.269
C08462=1012.612,313.297,-148.852,169.697,52.885,160.269
C08463=1012.618,313.544,-148.884,169.704,52.879,160.269
C08464=1012.624,313.792,-148.916,169.710,52.873,160.269
C08465=1012.630,314.040,-148.948,169.717,52.868,160.269
C08466=1012.636,314.288,-148.982,169.724,52.862,160.269
C08467=1012.641,314.535,-149.013,169.730,52.856,160.269
C08468=1012.647,314.783,-149.046,169.737,52.850,160.269
C08469=1012.654,315.030,-149.079,169.744,52.844,160.269
C08470=1012.660,315.279,-149.111,169.751,52.838,160.269
C08471=1012.666,315.526,-149.144,169.757,52.832,160.269
C08472=1012.671,315.774,-149.177,169.764,52.826,160.269
C08473=1012.677,316.022,-149.209,169.770,52.820,160.269
C08474=1012.683,316.269,-149.241,169.778,52.814,160.269
C08475=1012.689,316.517,-149.274,169.784,52.809,160.269
C08476=1012.695,316.765,-149.306,169.792,52.803,160.269
C08477=1012.702,317.013,-149.339,169.798,52.797,160.269
C08478=1012.707,317.261,-149.372,169.805,52.791,160.269
C08479=1012.713,317.508,-149.405,169.812,52.786,160.269
C08480=1012.719,317.756,-149.437,169.819,52.780,160.269
C08481=1012.726,318.004,-149.470,169.825,52.774,160.269
C08482=1012.732,318.252,-149.503,169.832,52.768,160.269
C08483=1012.738,318.500,-149.536,169.839,52.763,160.269
C08484=1012.744,318.747,-149.569,169.846,52.757,160.269
C08485=1012.750,318.995,-149.601,169.853,52.751,160.269
C08486=1012.756,319.242,-149.634,169.860,52.746,160.269
C08487=1012.763,319.490,-149.667,169.867,52.740,160.269
C08488=1012.769,319.737,-149.700,169.874,52.734,160.269
C08489=1012.775,319.986,-149.733,169.881,52.728,160.270
C08490=1012.782,320.234,-149.766,169.888,52.723,160.270
C08491=1012.788,320.481,-149.799,169.895,52.717,160.270
C08492=1012.794,320.729,-149.832,169.902,52.712,160.270
C08493=1012.800,320.976,-149.864,169.909,52.705,160.270
C08494=1012.806,321.224,-149.898,169.916,52.700,160.270
C08495=1012.812,321.472,-149.930,169.923,52.694,160.270
C08496=1012.819,321.720,-149.963,169.929,52.689,160.270
C08497=1012.825,321.968,-149.996,169.937,52.683,160.270
C08498=1012.832,322.215,-150.029,169.943,52.678,160.270
C08499=1012.837,322.463,-150.062,169.951,52.672,160.270
C08500=1012.844,322.711,-150.095,169.957,52.667,160.270
C08501=1012.851,323.013,-150.136,169.967,52.660,160.271
C08502=1012.859,323.316,-150.176,169.975,52.654,160.271
C08503=1012.868,323.618,-150.217,169.984,52.646,160.271
C08504=1012.875,323.921,-150.257,169.992,52.640,160.271
C08505=1012.883,324.169,-150.291,170.000,52.634,160.271
C08506=1012.888,324.417,-150.324,170.006,52.629,160.271
C08507=1012.894,324.665,-150.357,170.013,52.623,160.271
C08508=1012.901,324.913,-150.390,170.021,52.618,160.271
C08509=1012.908,325.160,-150.423,170.028,52.612,160.272
C08510=1012.914,325.407,-150.456,170.035,52.606,160.272
C08511=1012.921,325.655,-150.491,170.042,52.601,160.272
C08512=1012.927,325.903,-150.523,170.049,52.596,160.272
C08513=1012.933,326.150,-150.557,170.056,52.591,160.272
C08514=1012.939,326.398,-150.592,170.064,52.585,160.272
C08515=1012.946,326.645,-150.625,170.071,52.580,160.272
C08516=1012.951,326.893,-150.659,170.078,52.575,160.273
C08517=1012.958,327.141,-150.693,170.085,52.570,160.273
C08518=1012.964,327.388,-150.726,170.093,52.564,160.273
C08519=1012.971,327.636,-150.761,170.099,52.559,160.273
C08520=1012.977,327.884,-150.794,170.107,52.554,160.273
C08521=1012.984,328.132,-150.828,170.115,52.549,160.274
C08522=1012.990,328.379,-150.862,170.121,52.544,160.274
C08523=1012.997,328.627,-150.896,170.129,52.538,160.274
C08524=1013.003,328.874,-150.930,170.136,52.533,160.274
C08525=1013.009,329.122,-150.964,170.143,52.528,160.274
C08526=1013.015,329.370,-150.997,170.150,52.523,160.274
C08527=1013.022,329.618,-151.032,170.158,52.517,160.275
C08528=1013.028,329.865,-151.066,170.164,52.512,160.275
C08529=1013.035,330.112,-151.099,170.172,52.507,160.275
C08530=1013.041,330.360,-151.133,170.180,52.501,160.275
C08531=1013.047,330.608,-151.168,170.186,52.496,160.275
C08532=1013.054,330.855,-151.202,170.195,52.492,160.276
C08533=1013.060,331.103,-151.236,170.201,52.486,160.276
C08534=1013.067,331.351,-151.270,170.209,52.481,160.276
C08535=1013.074,331.598,-151.305,170.216,52.476,160.276
C08536=1013.080,331.845,-151.339,170.223,52.471,160.277
C08537=1013.087,332.093,-151.373,170.232,52.466,160.277
C08538=1013.093,332.341,-151.408,170.238,52.461,160.277
C08539=1013.099,332.588,-151.442,170.246,52.455,160.277
C08540=1013.106,332.836,-151.477,170.253,52.451,160.278
C08541=1013.113,333.083,-151.511,170.261,52.446,160.278
C08542=1013.119,333.330,-151.545,170.268,52.441,160.278
C08543=1013.126,333.578,-151.580,170.276,52.436,160.279
C08544=1013.132,333.826,-151.614,170.283,52.430,160.279
C08545=1013.139,334.073,-151.649,170.290,52.426,160.279
C08546=1013.145,334.321,-151.683,170.298,52.421,160.279
C08547=1013.151,334.568,-151.719,170.305,52.416,160.280
C08548=1013.158,334.816,-151.753,170.313,52.411,160.280
C08549=1013.165,335.063,-151.788,170.320,52.407,160.280
C08550=1013.171,335.311,-151.823,170.328,52.401,160.281
C08551=1013.177,335.558,-151.857,170.336,52.396,160.281
C08552=1013.184,335.806,-151.891,170.342,52.391,160.281
C08553=1013.191,336.053,-151.926,170.351,52.387,160.282
C08554=1013.198,336.301,-151.961,170.358,52.382,160.282
C08555=1013.204,336.548,-151.996,170.365,52.377,160.282
C08556=1013.211,336.796,-152.031,170.374,52.372,160.283
C08557=1013.218,337.044,-152.065,170.381,52.368,160.283
C08558=1013.224,337.291,-152.101,170.388,52.362,160.283
C08559=1013.231,337.538,-152.136,170.397,52.358,160.284
C08560=1013.238,337.786,-152.171,170.404,52.353,160.284
C08561=1013.246,338.084,-152.212,170.413,52.347,160.284
C08562=1013.254,338.383,-152.254,170.422,52.341,160.285
C08563=1013.262,338.681,-152.297,170.431,52.335,160.285
C08564=1013.270,338.979,-152.339,170.441,52.330,160.286
C08565=1013.276,339.227,-152.374,170.448,52.326,160.286
C08566=1013.283,339.474,-152.409,170.456,52.321,160.286
C08567=1013.289,339.722,-152.445,170.464,52.315,160.287
C08568=1013.296,339.968,-152.480,170.471,52.311,160.287
C08569=1013.304,340.216,-152.516,170.479,52.306,160.287
C08570=1013.311,340.464,-152.551,170.486,52.302,160.288
C08571=1013.317,340.711,-152.587,170.494,52.297,160.288
C08572=1013.323,340.959,-152.622,170.502,52.293,160.289
C08573=1013.330,341.206,-152.657,170.510,52.288,160.289
C08574=1013.337,341.454,-152.692,170.518,52.283,160.289
C08575=1013.344,341.701,-152.727,170.526,52.279,160.290
C08576=1013.351,341.948,-152.763,170.533,52.274,160.290
C08577=1013.357,342.196,-152.799,170.541,52.270,160.291
C08578=1013.364,342.443,-152.834,170.549,52.265,160.291
C08579=1013.371,342.690,-152.870,170.557,52.261,160.292
C08580=1013.378,342.937,-152.905,170.565,52.256,160.292
C08581=1013.384,343.185,-152.941,170.573,52.252,160.292
C08582=1013.392,343.433,-152.977,170.580,52.247,160.293
C08583=1013.399,343.680,-153.012,170.588,52.243,160.293
C08584=1013.406,343.927,-153.048,170.596,52.238,160.294
C08585=1013.412,344.174,-153.084,170.604,52.234,160.294
C08586=1013.419,344.422,-153.120,170.612,52.229,160.295
C08587=1013.426,344.669,-153.155,170.620,52.225,160.295
C08588=1013.433,344.916,-153.191,170.629,52.221,160.296
C08589=1013.440,345.164,-153.227,170.636,52.216,160.296
C08590=1013.447,345.411,-153.263,170.644,52.212,160.297
C08591=1013.454,345.658,-153.298,170.652,52.207,160.297
C08592=1013.461,345.906,-153.335,170.660,52.203,160.298
C08593=1013.467,346.154,-153.370,170.668,52.198,160.298
C08594=1013.475,346.401,-153.406,170.676,52.194,160.299
C08595=1013.481,346.648,-153.443,170.685,52.190,160.299
C08596=1013.488,346.895,-153.479,170.692,52.186,160.300
C08597=1013.495,347.143,-153.516,170.700,52.181,160.300
C08598=1013.502,347.390,-153.551,170.709,52.177,160.301
C08599=1013.510,347.637,-153.587,170.716,52.173,160.301
C08600=1013.516,347.884,-153.623,170.724,52.169,160.302
C08601=1013.523,348.132,-153.660,170.733,52.164,160.302
C08602=1013.530,348.379,-153.696,170.741,52.160,160.303
C08603=1013.537,348.627,-153.733,170.748,52.155,160.303
C08604=1013.544,348.873,-153.769,170.757,52.151,160.304
C08605=1013.551,349.121,-153.805,170.765,52.147,160.304
C08606=1013.558,349.368,-153.841,170.774,52.143,160.305
C08607=1013.565,349.616,-153.878,170.781,52.139,160.305
C08608=1013.572,349.862,-153.914,170.790,52.135,160.306
C08609=1013.579,350.110,-153.952,170.798,52.131,160.307
C08610=1013.587,350.357,-153.988,170.806,52.126,160.307
C08611=1013.593,350.604,-154.024,170.814,52.122,160.308
C08612=1013.601,350.851,-154.060,170.822,52.118,160.308
C08613=1013.608,351.099,-154.097,170.831,52.114,160.309
C08614=1013.615,351.345,-154.134,170.840,52.110,160.310
C08615=1013.622,351.593,-154.171,170.848,52.105,160.310
C08616=1013.630,351.841,-154.207,170.855,52.102,160.311
C08617=1013.637,352.087,-154.244,170.864,52.098,160.311
C08618=1013.644,352.334,-154.280,170.872,52.094,160.312
C08619=1013.651,352.582,-154.317,170.881,52.089,160.313
C08620=1013.659,352.829,-154.354,170.889,52.085,160.313
C08621=1013.667,353.126,-154.398,170.899,52.081,160.314
C08622=1013.676,353.420,-154.442,170.910,52.076,160.315
C08623=1013.685,353.716,-154.486,170.919,52.071,160.315
C08624=1013.693,354.012,-154.530,170.929,52.066,160.316
C08625=1013.701,354.259,-154.567,170.938,52.062,160.317
C08626=1013.708,354.506,-154.605,170.947,52.059,160.318
C08627=1013.715,354.754,-154.642,170.954,52.055,160.318
C08628=1013.722,355.000,-154.678,170.963,52.051,160.319
C08629=1013.729,355.247,-154.716,170.971,52.047,160.319
C08630=1013.736,355.495,-154.753,170.980,52.043,160.320
C08631=1013.744,355.742,-154.790,170.989,52.039,160.321
C08632=1013.752,355.989,-154.827,170.998,52.035,160.322
C08633=1013.759,356.236,-154.865,171.006,52.031,160.322
C08634=1013.766,356.483,-154.902,171.014,52.028,160.323
C08635=1013.774,356.730,-154.939,171.023,52.024,160.324
C08636=1013.781,356.977,-154.977,171.031,52.020,160.324
C08637=1013.788,357.225,-155.013,171.040,52.016,160.325
C08638=1013.795,357.472,-155.051,171.049,52.013,160.326
C08639=1013.803,357.719,-155.088,171.057,52.008,160.326
C08640=1013.811,357.966,-155.126,171.066,52.004,160.327
C08641=1013.818,358.213,-155.164,171.075,52.001,160.328
C08642=1013.826,358.460,-155.201,171.083,51.997,160.329
C08643=1013.833,358.707,-155.239,171.092,51.993,160.329
C08644=1013.840,358.954,-155.276,171.101,51.989,160.330
C08645=1013.847,359.201,-155.314,171.109,51.986,160.331
C08646=1013.855,359.448,-155.352,171.118,51.983,160.332
C08647=1013.863,359.696,-155.390,171.126,51.979,160.332
C08648=1013.870,359.943,-155.427,171.135,51.975,160.333
C08649=1013.877,360.189,-155.466,171.144,51.972,160.334
C08650=1013.885,360.436,-155.503,171.153,51.968,160.335
C08651=1013.892,360.683,-155.541,171.162,51.964,160.336
C08652=1013.899,360.930,-155.579,171.171,51.961,160.336
C08653=1013.907,361.178,-155.617,171.179,51.957,160.337
C08654=1013.915,361.424,-155.655,171.188,51.954,160.338
C08655=1013.922,361.672,-155.693,171.197,51.950,160.339
C08656=1013.930,361.918,-155.731,171.206,51.947,160.340
C08657=1013.938,362.165,-155.769,171.215,51.943,160.340
C08658=1013.945,362.412,-155.807,171.224,51.939,160.341
C08659=1013.953,362.659,-155.845,171.233,51.936,160.342
C08660=1013.961,362.906,-155.884,171.242,51.932,160.343
C08661=1013.968,363.153,-155.921,171.251,51.929,160.344
C08662=1013.976,363.400,-155.960,171.260,51.925,160.344
C08663=1013.984,363.647,-155.998,171.269,51.922,160.345
C08664=1013.991,363.894,-156.036,171.278,51.919,160.346
C08665=1013.999,364.141,-156.074,171.287,51.915,160.347
C08666=1014.006,364.388,-156.113,171.296,51.912,160.348
C08667=1014.013,364.635,-156.151,171.305,51.908,160.349
C08668=1014.022,364.882,-156.190,171.314,51.905,160.350
C08669=1014.029,365.128,-156.228,171.323,51.901,160.350
C08670=1014.037,365.376,-156.267,171.332,51.898,160.351
C08671=1014.045,365.622,-156.305,171.342,51.894,160.352
C08672=1014.053,365.869,-156.344,171.351,51.891,160.353
C08673=1014.061,366.116,-156.382,171.360,51.888,160.354
C08674=1014.069,366.363,-156.421,171.369,51.885,160.355
C08675=1014.077,366.610,-156.459,171.378,51.881,160.356
C08676=1014.084,366.857,-156.497,171.387,51.878,160.357
C08677=1014.093,367.104,-156.536,171.396,51.875,160.358
C08678=1014.099,367.351,-156.575,171.405,51.872,160.359
C08679=1014.108,367.597,-156.614,171.416,51.868,160.360
C08680=1014.115,367.844,-156.652,171.425,51.865,160.361
C08681=1014.126,368.148,-156.701,171.436,51.861,160.362
C08682=1014.135,368.451,-156.749,171.447,51.857,160.363
C08683=1014.144,368.754,-156.797,171.458,51.854,160.364
C08684=1014.154,369.057,-156.845,171.470,51.849,160.365
C08685=1014.161,369.305,-156.884,171.480,51.846,160.366
C08686=1014.170,369.551,-156.923,171.489,51.843,160.367
C08687=1014.178,369.799,-156.962,171.498,51.840,160.368
C08688=1014.185,370.045,-157.001,171.507,51.837,160.369
C08689=1014.193,370.292,-157.040,171.517,51.833,160.370
C08690=1014.202,370.539,-157.079,171.527,51.831,160.371
C08691=1014.209,370.785,-157.119,171.536,51.828,160.372
C08692=1014.218,371.032,-157.159,171.545,51.824,160.373
C08693=1014.225,371.279,-157.197,171.555,51.822,160.374
C08694=1014.233,371.525,-157.237,171.565,51.818,160.376
C08695=1014.241,371.772,-157.276,171.574,51.816,160.377
C08696=1014.249,372.019,-157.316,171.583,51.812,160.377
C08697=1014.258,372.266,-157.355,171.593,51.809,160.378
C08698=1014.266,372.513,-157.394,171.603,51.806,160.380
C08699=1014.273,372.760,-157.434,171.613,51.803,160.381
C08700=1014.282,373.006,-157.473,171.622,51.801,160.382
C08701=1014.290,373.253,-157.512,171.632,51.797,160.383
C08702=1014.298,373.500,-157.552,171.642,51.795,160.384
C08703=1014.307,373.746,-157.592,171.651,51.792,160.385
C08704=1014.315,373.993,-157.631,171.661,51.789,160.386
C08705=1014.323,374.240,-157.671,171.671,51.786,160.387
C08706=1014.332,374.486,-157.711,171.680,51.783,160.388
C08707=1014.339,374.733,-157.751,171.691,51.780,160.389
C08708=1014.348,374.979,-157.790,171.700,51.777,160.391
C08709=1014.356,375.226,-157.830,171.709,51.774,160.392
C08710=1014.364,375.473,-157.869,171.720,51.771,160.393
C08711=1014.372,375.719,-157.910,171.729,51.768,160.394
C08712=1014.381,375.966,-157.950,171.739,51.766,160.395
C08713=1014.389,376.213,-157.990,171.749,51.763,160.396
C08714=1014.397,376.460,-158.030,171.759,51.760,160.397
C08715=1014.405,376.706,-158.071,171.770,51.757,160.399
C08716=1014.413,376.952,-158.110,171.779,51.755,160.400
C08717=1014.421,377.199,-158.151,171.788,51.752,160.401
C08718=1014.430,377.446,-158.192,171.799,51.749,160.402
C08719=1014.438,377.692,-158.231,171.809,51.747,160.403
C08720=1014.446,377.939,-158.272,171.819,51.744,160.405
C08721=1014.454,378.185,-158.313,171.829,51.741,160.406
C08722=1014.463,378.432,-158.354,171.840,51.739,160.407
C08723=1014.471,378.679,-158.393,171.849,51.736,160.408
C08724=1014.479,378.925,-158.433,171.860,51.733,160.409
C08725=1014.488,379.172,-158.474,171.869,51.730,160.411
C08726=1014.497,379.418,-158.515,171.880,51.728,160.412
C08727=1014.505,379.665,-158.556,171.890,51.726,160.413
C08728=1014.514,379.911,-158.596,171.900,51.722,160.414
C08729=1014.522,380.157,-158.637,171.910,51.720,160.416
C08730=1014.531,380.404,-158.677,171.921,51.718,160.417
C08731=1014.539,380.650,-158.718,171.930,51.715,160.418
C08732=1014.548,380.897,-158.759,171.941,51.712,160.419
C08733=1014.556,381.143,-158.799,171.951,51.710,160.421
C08734=1014.565,381.390,-158.840,171.962,51.708,160.422
C08735=1014.573,381.636,-158.881,171.971,51.705,160.423
C08736=1014.582,381.883,-158.921,171.982,51.702,160.424
C08737=1014.591,382.130,-158.963,171.992,51.700,160.426
C08738=1014.599,382.376,-159.003,172.002,51.697,160.427
C08739=1014.608,382.623,-159.044,172.013,51.695,160.428
C08740=1014.617,382.869,-159.084,172.024,51.692,160.430
C08741=1014.626,383.115,-159.126,172.034,51.690,160.431
C08742=1014.635,383.360,-159.167,172.044,51.687,160.432
C08743=1014.647,383.696,-159.222,172.059,51.684,160.434
C08744=1014.658,384.029,-159.278,172.073,51.681,160.436
C08745=1014.670,384.365,-159.333,172.087,51.678,160.438
C08746=1014.682,384.699,-159.390,172.102,51.675,160.440
C08747=1014.691,384.946,-159.431,172.112,51.672,160.441
C08748=1014.700,385.193,-159.472,172.123,51.670,160.443
C08749=1014.709,385.439,-159.514,172.134,51.668,160.444
C08750=1014.717,385.685,-159.555,172.144,51.666,160.446
C08751=1014.726,385.931,-159.597,172.155,51.663,160.447
C08752=1014.735,386.177,-159.639,172.166,51.661,160.448
C08753=1014.744,386.424,-159.680,172.177,51.659,160.450
C08754=1014.753,386.670,-159.722,172.188,51.657,160.451
C08755=1014.761,386.917,-159.763,172.198,51.654,160.453
C08756=1014.770,387.163,-159.805,172.209,51.652,160.454
C08757=1014.779,387.410,-159.847,172.220,51.650,160.456
C08758=1014.789,387.655,-159.889,172.231,51.648,160.457
C08759=1014.798,387.902,-159.931,172.242,51.645,160.459
C08760=1014.806,388.148,-159.972,172.252,51.644,160.460
C08761=1014.815,388.395,-160.014,172.263,51.642,160.462
C08762=1014.824,388.641,-160.056,172.274,51.640,160.463
C08763=1014.834,388.887,-160.098,172.285,51.637,160.465
C08764=1014.842,389.133,-160.140,172.296,51.635,160.466
C08765=1014.851,389.380,-160.182,172.308,51.633,160.468
C08766=1014.860,389.625,-160.225,172.319,51.631,160.469
C08767=1014.869,389.872,-160.267,172.330,51.629,160.471
C08768=1014.878,390.118,-160.309,172.341,51.627,160.472
C08769=1014.887,390.364,-160.351,172.352,51.625,160.474
C08770=1014.897,390.610,-160.393,172.362,51.623,160.475
C08771=1014.906,390.857,-160.435,172.373,51.621,160.477
C08772=1014.915,391.102,-160.478,172.385,51.619,160.479
C08773=1014.924,391.349,-160.519,172.396,51.617,160.480
C08774=1014.934,391.595,-160.562,172.407,51.615,160.482
C08775=1014.942,391.841,-160.605,172.418,51.613,160.483
C08776=1014.952,392.087,-160.648,172.430,51.612,160.485
C08777=1014.960,392.333,-160.689,172.442,51.609,160.487
C08778=1014.970,392.580,-160.733,172.453,51.608,160.488
C08779=1014.979,392.826,-160.775,172.464,51.606,160.490
C08780=1014.988,393.072,-160.818,172.476,51.604,160.492
C08781=1014.998,393.318,-160.860,172.487,51.602,160.493
C08782=1015.006,393.564,-160.903,172.498,51.600,160.495
C08783=1015.016,393.811,-160.946,172.510,51.599,160.497
C08784=1015.025,394.056,-160.989,172.521,51.597,160.498
C08785=1015.036,394.302,-161.032,172.533,51.595,160.500
C08786=1015.044,394.548,-161.075,172.544,51.593,160.502
C08787=1014.693,392.504,-161.065,172.432,51.670,160.501
C08788=1014.684,392.258,-161.023,172.420,51.672,160.499
C08789=1014.675,392.012,-160.981,172.409,51.674,160.498
C08790=1014.666,391.766,-160.938,172.398,51.676,160.496
C08791=1014.656,391.520,-160.895,172.387,51.678,160.495
C08792=1014.648,391.273,-160.853,172.375,51.680,160.493
C08793=1014.638,391.028,-160.811,172.364,51.682,160.491
C08794=1014.629,390.781,-160.769,172.353,51.684,160.490
C08795=1014.620,390.535,-160.726,172.342,51.686,160.488
C08796=1014.611,390.288,-160.684,172.331,51.688,160.487
C08797=1014.601,390.043,-160.642,172.319,51.690,160.485
C08798=1014.592,389.796,-160.600,172.309,51.693,160.484
C08799=1014.583,389.551,-160.558,172.297,51.695,160.482
C08800=1014.575,389.304,-160.515,172.286,51.697,160.481
C08801=1014.566,389.058,-160.474,172.275,51.699,160.479
C08802=1014.557,388.812,-160.431,172.264,51.701,160.478
C08803=1014.548,388.565,-160.390,172.253,51.703,160.476
C08804=1014.539,388.319,-160.348,172.242,51.705,160.474
C08805=1014.530,388.073,-160.306,172.232,51.707,160.473
C08806=1014.521,387.826,-160.264,172.221,51.709,160.472
C08807=1014.512,387.580,-160.223,172.210,51.712,160.470
C08808=1014.503,387.334,-160.181,172.199,51.714,160.469
C08809=1014.494,387.087,-160.139,172.188,51.717,160.467
C08810=1014.485,386.841,-160.098,172.177,51.719,160.466
C08811=1014.476,386.594,-160.056,172.166,51.721,160.464
C08812=1014.467,386.348,-160.014,172.156,51.723,160.463
C08813=1014.459,386.102,-159.972,172.145,51.725,160.461
C08814=1014.450,385.855,-159.931,172.134,51.728,160.460
C08815=1014.441,385.610,-159.889,172.123,51.730,160.458
C08816=1014.433,385.363,-159.848,172.112,51.732,160.457
C08817=1014.424,385.116,-159.807,172.102,51.735,160.456
C08818=1014.415,384.870,-159.765,172.091,51.737,160.454
C08819=1014.407,384.624,-159.724,172.080,51.739,160.453
C08820=1014.399,384.414,-159.689,172.072,51.742,160.452
C08821=1014.391,384.204,-159.654,172.062,51.744,160.451
C08822=1014.384,383.995,-159.619,172.053,51.746,160.449
C08823=1014.376,383.784,-159.584,172.044,51.748,160.448
C08824=1014.369,383.575,-159.549,172.035,51.750,160.447
C08825=1014.361,383.366,-159.514,172.026,51.752,160.446
C08826=1014.354,383.156,-159.480,172.017,51.754,160.445
C08827=1014.346,382.946,-159.445,172.009,51.756,160.444
C08828=1014.338,382.700,-159.404,171.998,51.758,160.442
C08829=1014.329,382.453,-159.362,171.987,51.762,160.441
C08830=1014.320,382.208,-159.322,171.978,51.764,160.440
C08831=1014.312,381.961,-159.281,171.967,51.766,160.438
C08832=1014.303,381.714,-159.240,171.956,51.769,160.437
C08833=1014.294,381.468,-159.200,171.946,51.771,160.436
C08834=1014.286,381.221,-159.159,171.935,51.774,160.434
C08835=1014.278,380.974,-159.119,171.925,51.777,160.433
C08836=1014.268,380.728,-159.078,171.915,51.779,160.432
C08837=1014.260,380.481,-159.038,171.904,51.782,160.431
C08838=1014.252,380.235,-158.997,171.895,51.785,160.430
C08839=1014.243,379.988,-158.956,171.884,51.787,160.428
C08840=1014.235,379.742,-158.916,171.873,51.790,160.427
C08841=1014.226,379.495,-158.875,171.864,51.793,160.426
C08842=1014.218,379.249,-158.834,171.853,51.795,160.424
C08843=1014.209,379.003,-158.794,171.844,51.798,160.423
C08844=1014.201,378.756,-158.753,171.833,51.801,160.422
C08845=1014.193,378.509,-158.713,171.824,51.803,160.421
C08846=1014.184,378.263,-158.673,171.813,51.806,160.420
C08847=1014.176,378.016,-158.632,171.803,51.809,160.418
C08848=1014.168,377.769,-158.592,171.793,51.811,160.417
C08849=1014.160,377.523,-158.552,171.783,51.814,160.416
C08850=1014.151,377.277,-158.512,171.773,51.817,160.415
C08851=1014.143,377.030,-158.472,171.763,51.819,160.414
C08852=1014.135,376.783,-158.431,171.753,51.823,160.412
C08853=1014.126,376.536,-158.391,171.743,51.826,160.411
C08854=1014.118,376.290,-158.351,171.732,51.828,160.410
C08855=1014.111,376.043,-158.311,171.723,51.831,160.409
C08856=1014.102,375.797,-158.270,171.714,51.834,160.408
C08857=1014.094,375.550,-158.231,171.703,51.837,160.407
C08858=1014.086,375.304,-158.190,171.694,51.840,160.406
C08859=1014.078,375.057,-158.150,171.684,51.843,160.404
C08860=1014.070,374.810,-158.111,171.674,51.846,160.403
C08861=1014.061,374.563,-158.071,171.664,51.849,160.402
C08862=1014.053,374.316,-158.031,171.654,51.852,160.401
C08863=1014.045,374.070,-157.992,171.645,51.855,160.400
C08864=1014.036,373.823,-157.953,171.635,51.858,160.399
C08865=1014.028,373.576,-157.913,171.625,51.861,160.398
C08866=1014.020,373.330,-157.874,171.615,51.864,160.397
C08867=1014.011,373.083,-157.834,171.605,51.867,160.396
C08868=1014.004,372.836,-157.794,171.596,51.869,160.395
C08869=1013.995,372.589,-157.755,171.586,51.873,160.393
C08870=1013.987,372.344,-157.716,171.576,51.875,160.392
C08871=1013.980,372.097,-157.676,171.567,51.879,160.392
C08872=1013.972,371.849,-157.638,171.557,51.882,160.390
C08873=1013.964,371.603,-157.598,171.547,51.885,160.389
C08874=1013.955,371.356,-157.558,171.538,51.888,160.388
C08875=1013.947,371.109,-157.519,171.529,51.891,160.387
C08876=1013.940,370.862,-157.480,171.519,51.894,160.386
C08877=1013.932,370.616,-157.441,171.510,51.898,160.385
C08878=1013.923,370.369,-157.401,171.500,51.901,160.384
C08879=1013.916,370.122,-157.362,171.490,51.904,160.383
C08880=1013.907,369.875,-157.323,171.481,51.907,160.382
C08881=1013.901,369.628,-157.284,171.472,51.910,160.381
C08882=1013.892,369.382,-157.245,171.463,51.913,160.380
C08883=1013.884,369.135,-157.206,171.453,51.916,160.379
C08884=1013.874,368.829,-157.158,171.441,51.921,160.378
C08885=1013.864,368.524,-157.109,171.430,51.924,160.377
C08886=1013.855,368.218,-157.060,171.418,51.929,160.376
C08887=1013.846,367.912,-157.013,171.407,51.933,160.374
C08888=1013.838,367.666,-156.974,171.398,51.936,160.374
C08889=1013.830,367.419,-156.935,171.388,51.939,160.373
C08890=1013.822,367.171,-156.896,171.378,51.943,160.372
C08891=1013.815,366.925,-156.857,171.369,51.946,160.371
C08892=1013.806,366.678,-156.818,171.360,51.949,160.370
C08893=1013.799,366.432,-156.780,171.351,51.952,160.369
C08894=1013.791,366.185,-156.741,171.342,51.956,160.368
C08895=1013.783,365.938,-156.703,171.333,51.959,160.367
C08896=1013.775,365.691,-156.665,171.323,51.963,160.366
C08897=1013.768,365.444,-156.627,171.314,51.966,160.365
C08898=1013.760,365.196,-156.588,171.305,51.970,160.364
C08899=1013.752,364.950,-156.550,171.296,51.973,160.364
C08900=1013.744,364.709,-156.513,171.287,51.977,160.363
C08901=1013.738,364.468,-156.475,171.278,51.980,160.362
C08902=1013.730,364.228,-156.438,171.269,51.984,160.361
C08903=1013.722,363.987,-156.401,171.260,51.987,160.360
C08904=1013.715,363.747,-156.364,171.252,51.990,160.359
C08905=1013.707,363.506,-156.326,171.243,51.994,160.359
C08906=1013.699,363.266,-156.289,171.234,51.997,160.358
C08907=1013.692,363.025,-156.252,171.225,52.000,160.357
C08908=1013.684,362.778,-156.213,171.216,52.004,160.356
C08909=1013.677,362.531,-156.176,171.208,52.008,160.355
C08910=1013.669,362.284,-156.138,171.199,52.011,160.354
C08911=1013.662,362.038,-156.099,171.190,52.015,160.354
C08912=1013.654,361.790,-156.061,171.181,52.018,160.353
C08913=1013.646,361.544,-156.023,171.172,52.022,160.352
C08914=1013.639,361.296,-155.986,171.163,52.026,160.351
C08915=1013.632,361.050,-155.947,171.154,52.029,160.350
C08916=1013.624,360.803,-155.910,171.145,52.033,160.349
C08917=1013.617,360.555,-155.872,171.137,52.037,160.349
